# B&R Automation Studio project NAELD004C00R10L518F00 (part 23)

#### Act_Main_Bffr.st
```iecst
(** 2013-05-27 **)
ACTION Act_Main_Bffr:

	CASE usiStep OF
		//Buffer 1
		0:
			eBuffer1Act	:= BufferActCreateDir;

			IF (p_eBuffer1Status = Done) AND (p_eBuffer1Stat = BufferActCreateDir) THEN

				eBuffer1Act	:= BufferActIdle;
				usiStep		:= 1;

			ELSIF p_eBuffer1Status = Error THEN

				eBuffer1Act	:= BufferActIdle;
				usiStep		:= 10;

			END_IF

		1:
			eBuffer1Act	:= BufferActBGStartBffrSetFull;		//BufferActBGStartBffrSetMty

			IF (p_eBuffer1Status = Done) AND (p_eBuffer1Stat = BufferActBGStartBffrSetFull) THEN		//BufferActBGStartBffrSetMty

				eBuffer1Act	:= BufferActIdle;
				usiStep		:= 2;

			ELSIF p_eBuffer1Status = Error THEN

				eBuffer1Act	:= BufferActIdle;
				usiStep		:= 10;

			END_IF

		2:
			IF p_bMagPresent1 = FALSE AND p_bMagPresentSensor1 = TRUE THEN
				usiStep	:= 4;
			ELSE
				usiStep	:= 3;
			END_IF

		3:
			eBuffer1Act	:= BufferActBGStartUpdtSen;

			IF (p_eBuffer1Status = Done) AND (p_eBuffer1Stat = BufferActBGStartUpdtSen) THEN

				eBuffer1Act	:= BufferActIdle;
				usiStep		:= 5;

			ELSIF p_eBuffer1Status = Error THEN

				eBuffer1Act	:= BufferActIdle;
				usiStep		:= 10;

			END_IF

		4:
			eBuffer1Act	:= BufferActBGStartUpdtSen;

			IF (p_eBuffer1Status = Done) AND (p_eBuffer1Stat = BufferActBGStartUpdtSen) THEN

				eBuffer1Act	:= BufferActIdle;
				usiStep		:= 6;

			ELSIF p_eBuffer1Status = Error THEN

				eBuffer1Act	:= BufferActIdle;
				usiStep		:= 10;

			END_IF

		5:
			eBuffer1Act	:= BufferActGetRetainBffr;

			IF (p_eBuffer1Status = Done) AND (p_eBuffer1Stat = BufferActGetRetainBffr) THEN

				eBuffer1Act	:= BufferActIdle;
				usiStep		:= 7;

			ELSIF p_eBuffer1Status = Error THEN

				eBuffer1Act	:= BufferActIdle;
				usiStep		:= 10;

			END_IF

		6:
			eBuffer1Act	:= BufferActSetFull;		//BufferActSetMty

			IF (p_eBuffer1Status = Done) AND (p_eBuffer1Stat = BufferActSetFull) THEN		//BufferActSetMty

				eBuffer1Act	:= BufferActIdle;
				usiStep		:= 7;

			ELSIF p_eBuffer1Status = Error THEN

				eBuffer1Act	:= BufferActIdle;
				usiStep		:= 10;

			END_IF

		7:
			eBuffer1Act	:= BufferActBGStartCoolFan;

			IF (p_eBuffer1Status = Done) AND (p_eBuffer1Stat = BufferActBGStartCoolFan) THEN

				eBuffer1Act		:= BufferActIdle;
				usiStep			:= 10;

			ELSIF p_eBuffer1Status = Error THEN

				eBuffer1Act		:= BufferActIdle;
				usiStep			:= 10;

			END_IF

		//Buffer 2
		10:
			eBuffer2Act	:= BufferActCreateDir;

			IF (p_eBuffer2Status = Done) AND (p_eBuffer2Stat = BufferActCreateDir) THEN

				eBuffer2Act	:= BufferActIdle;
				usiStep		:= 11;

			ELSIF p_eBuffer2Status = Error THEN

				eBuffer2Act	:= BufferActIdle;
				usiStep		:= 20;

			END_IF

		11:
			eBuffer2Act	:= BufferActBGStartBffrSetFull;		//BufferActBGStartBffrSetMty

			IF (p_eBuffer2Status = Done) AND (p_eBuffer2Stat = BufferActBGStartBffrSetFull) THEN		//BufferActBGStartBffrSetMty

				eBuffer2Act	:= BufferActIdle;
				usiStep		:= 12;

			ELSIF p_eBuffer2Status = Error THEN

				eBuffer2Act	:= BufferActIdle;
				usiStep		:= 20;

			END_IF

		12:
			IF p_bMagPresent2 = FALSE AND p_bMagPresentSensor2 = TRUE THEN
				usiStep	:= 14;
			ELSE
				usiStep	:= 13;
			END_IF

		13:
			eBuffer2Act	:= BufferActBGStartUpdtSen;

			IF (p_eBuffer2Status = Done) AND (p_eBuffer2Stat = BufferActBGStartUpdtSen) THEN

				eBuffer2Act	:= BufferActIdle;
				usiStep		:= 15;

			ELSIF p_eBuffer2Status = Error THEN

				eBuffer2Act	:= BufferActIdle;
				usiStep		:= 20;

			END_IF

		14:
			eBuffer2Act	:= BufferActBGStartUpdtSen;

			IF (p_eBuffer2Status = Done) AND (p_eBuffer2Stat = BufferActBGStartUpdtSen) THEN

				eBuffer2Act	:= BufferActIdle;
				usiStep		:= 16;

			ELSIF p_eBuffer2Status = Error THEN

				eBuffer2Act	:= BufferActIdle;
				usiStep		:= 20;

			END_IF

		15:
			eBuffer2Act	:= BufferActGetRetainBffr;

			IF (p_eBuffer2Status = Done) AND (p_eBuffer2Stat = BufferActGetRetainBffr) THEN

				eBuffer2Act	:= BufferActIdle;
				usiStep		:= 17;

			ELSIF p_eBuffer2Status = Error THEN

				eBuffer2Act	:= BufferActIdle;
				usiStep		:= 20;

			END_IF

		16:
			eBuffer2Act	:= BufferActSetFull;		//BufferActSetMty

			IF (p_eBuffer2Status = Done) AND (p_eBuffer2Stat = BufferActSetFull) THEN		//BufferActSetMty

				eBuffer2Act	:= BufferActIdle;
				usiStep		:= 17;

			ELSIF p_eBuffer2Status = Error THEN

				eBuffer2Act	:= BufferActIdle;
				usiStep		:= 20;

			END_IF

		17:
			eBuffer2Act	:= BufferActBGStartCoolFan;

			IF (p_eBuffer2Status = Done) AND (p_eBuffer2Stat = BufferActBGStartCoolFan) THEN

				eBuffer2Act		:= BufferActIdle;
				usiStep			:= 20;

			ELSIF p_eBuffer2Status = Error THEN

				eBuffer2Act		:= BufferActIdle;
				usiStep			:= 20;

			END_IF

		//Buffer 3
		20:
			eBuffer3Act	:= BufferActCreateDir;

			IF (p_eBuffer3Status = Done) AND (p_eBuffer3Stat = BufferActCreateDir) THEN

				eBuffer3Act		:= BufferActIdle;
				usiStep			:= 21;

			ELSIF p_eBuffer3Status = Error THEN

				eBuffer3Act		:= BufferActIdle;
				usiStep			:= 30;

			END_IF

		21:
			eBuffer3Act	:= BufferActBGStartBffrSetFull;		//BufferActBGStartBffrSetMty

			IF (p_eBuffer3Status = Done) AND (p_eBuffer3Stat = BufferActBGStartBffrSetFull) THEN		//BufferActBGStartBffrSetMty

				eBuffer3Act		:= BufferActIdle;
				usiStep			:= 22;

			ELSIF p_eBuffer3Status = Error THEN

				eBuffer3Act		:= BufferActIdle;
				usiStep			:= 30;

			END_IF

		22:
			IF p_bMagPresent3 = FALSE AND p_bMagPresentSensor3 = TRUE THEN
				usiStep	:= 24;
			ELSE
				usiStep	:= 23;
			END_IF

		23:
			eBuffer3Act	:= BufferActBGStartUpdtSen;

			IF (p_eBuffer3Status = Done) AND (p_eBuffer3Stat = BufferActBGStartUpdtSen) THEN

				eBuffer3Act		:= BufferActIdle;
				usiStep			:= 25;

			ELSIF p_eBuffer3Status = Error THEN

				eBuffer3Act		:= BufferActIdle;
				usiStep			:= 30;

			END_IF

		24:
			eBuffer3Act	:= BufferActBGStartUpdtSen;

			IF (p_eBuffer3Status = Done) AND (p_eBuffer3Stat = BufferActBGStartUpdtSen) THEN

				eBuffer3Act		:= BufferActIdle;
				usiStep			:= 26;

			ELSIF p_eBuffer3Status = Error THEN

				eBuffer3Act		:= BufferActIdle;
				usiStep			:= 30;

			END_IF

		25:
			eBuffer3Act	:= BufferActGetRetainBffr;

			IF (p_eBuffer3Status = Done) AND (p_eBuffer3Stat = BufferActGetRetainBffr) THEN

				eBuffer3Act		:= BufferActIdle;
				usiStep			:= 27;

			ELSIF p_eBuffer3Status = Error THEN

				eBuffer3Act		:= BufferActIdle;
				usiStep			:= 30;

			END_IF

		26:
			eBuffer3Act	:= BufferActSetFull;		//BufferActSetMty

			IF (p_eBuffer3Status = Done) AND (p_eBuffer3Stat = BufferActSetFull) THEN		//BufferActSetMty

				eBuffer3Act		:= BufferActIdle;
				usiStep			:= 27;

			ELSIF p_eBuffer3Status = Error THEN

				eBuffer3Act		:= BufferActIdle;
				usiStep			:= 30;

			END_IF

		27:
			eBuffer3Act	:= BufferActBGStartCoolFan;

			IF (p_eBuffer3Status = Done) AND (p_eBuffer3Stat = BufferActBGStartCoolFan) THEN

				eBuffer3Act		:= BufferActIdle;
				usiStep			:= 30;

			ELSIF p_eBuffer3Status = Error THEN

				eBuffer3Act		:= BufferActIdle;
				usiStep			:= 30;

			END_IF

			//Buffer 4
		30:
			eBuffer4Act	:= BufferActCreateDir;

			IF (p_eBuffer4Status = Done) AND (p_eBuffer4Stat = BufferActCreateDir) THEN

				eBuffer4Act		:= BufferActIdle;
				usiStep			:= 31;

			ELSIF p_eBuffer4Status = Error THEN

				eBuffer4Act		:= BufferActIdle;
				usiStep			:= 0;
				eStartupStep1	:= StartupStepAlarm;

			END_IF

		31:
			eBuffer4Act	:= BufferActBGStartBffrSetFull;		//BufferActBGStartBffrSetMty

			IF (p_eBuffer4Status = Done) AND (p_eBuffer4Stat = BufferActBGStartBffrSetFull) THEN		//BufferActBGStartBffrSetMty

				eBuffer4Act		:= BufferActIdle;
				usiStep			:= 32;

			ELSIF p_eBuffer4Status = Error THEN

				eBuffer4Act		:= BufferActIdle;
				usiStep			:= 0;
				eStartupStep1	:= StartupStepAlarm;

			END_IF

		32:
			IF p_bMagPresent4 = FALSE AND p_bMagPresentSensor4 = TRUE THEN
				usiStep	:= 34;
			ELSE
				usiStep	:= 33;
			END_IF

		33:
			eBuffer4Act	:= BufferActBGStartUpdtSen;

			IF (p_eBuffer4Status = Done) AND (p_eBuffer4Stat = BufferActBGStartUpdtSen) THEN

				eBuffer4Act		:= BufferActIdle;
				usiStep			:= 35;

			ELSIF p_eBuffer4Status = Error THEN

				eBuffer4Act		:= BufferActIdle;
				usiStep			:= 0;
				eStartupStep1	:= StartupStepAlarm;

			END_IF

		34:
			eBuffer4Act	:= BufferActBGStartUpdtSen;

			IF (p_eBuffer4Status = Done) AND (p_eBuffer4Stat = BufferActBGStartUpdtSen) THEN

				eBuffer4Act		:= BufferActIdle;
				usiStep			:= 36;

			ELSIF p_eBuffer4Status = Error THEN

				eBuffer4Act		:= BufferActIdle;
				usiStep			:= 0;
				eStartupStep1	:= StartupStepAlarm;

			END_IF

		35:
			eBuffer4Act	:= BufferActGetRetainBffr;

			IF (p_eBuffer4Status = Done) AND (p_eBuffer4Stat = BufferActGetRetainBffr) THEN

				eBuffer4Act		:= BufferActIdle;
				usiStep			:= 37;

			ELSIF p_eBuffer4Status = Error THEN

				eBuffer4Act		:= BufferActIdle;
				usiStep			:= 0;
				eStartupStep1	:= StartupStepAlarm;

			END_IF

		36:
			eBuffer4Act	:= BufferActSetFull;		//BufferActSetMty

			IF (p_eBuffer4Status = Done) AND (p_eBuffer4Stat = BufferActSetFull) THEN		//BufferActSetMty

				eBuffer4Act		:= BufferActIdle;
				usiStep			:= 37;

			ELSIF p_eBuffer4Status = Error THEN

				eBuffer4Act		:= BufferActIdle;
				usiStep			:= 0;
				eStartupStep1	:= StartupStepAlarm;

			END_IF

		37:
			eBuffer4Act	:= BufferActBGStartCoolFan;

			IF (p_eBuffer4Status = Done) AND (p_eBuffer4Stat = BufferActBGStartCoolFan) THEN

				eBuffer4Act		:= BufferActIdle;
				usiStep			:= 0;
				eStartupStep1	:= StartupStepAlarm;

			ELSIF p_eBuffer4Status = Error THEN

				eBuffer4Act		:= BufferActIdle;
				usiStep			:= 0;
				eStartupStep1	:= StartupStepAlarm;

			END_IF
	END_CASE

END_ACTION
```

#### Act_Main_Alarm.st
```iecst
(** 2019-03-28 **)
ACTION Act_Main_Alarm:

	CASE usiStep OF
		0:
			eAlarmAct	:= AlarmActCreateDir;

			IF (p_eAlarmStatus = Done) AND (p_eAlarmStat = AlarmActCreateDir) THEN

				eAlarmAct		:= AlarmActIdle;
				usiStep			:= 1;

			ELSIF p_eAlarmStatus = Error THEN

				eAlarmAct		:= AlarmActIdle;
				usiStep			:= 0;
		//		eStartupStep1	:= StartupStepHermes;
				eStartupStep1	:= StartupStepSerial;
			END_IF

		1:
			eAlarmAct	:= AlarmActDeleteOldLog;

			IF (p_eAlarmStatus = Done) AND (p_eAlarmStat = AlarmActDeleteOldLog) THEN

				eAlarmAct		:= AlarmActIdle;
				usiStep			:= 2;

			ELSIF p_eAlarmStatus = Error THEN

				eAlarmAct		:= AlarmActIdle;
				usiStep			:= 0;
		//		eStartupStep1	:= StartupStepHermes;
				eStartupStep1	:= StartupStepSerial;
			END_IF

		2:
			eAlarmAct	:= AlarmActReadHistory;

			IF (p_eAlarmStatus = Done) AND (p_eAlarmStat = AlarmActReadHistory) THEN

				eAlarmAct		:= AlarmActIdle;
				usiStep			:= 3;

			ELSIF p_eAlarmStatus = Error THEN

				eAlarmAct		:= AlarmActIdle;
				usiStep			:= 0;
		//		eStartupStep1	:= StartupStepHermes;
				eStartupStep1	:= StartupStepSerial;
			END_IF

		3:
			eAlarmAct	:= AlarmActBGStartLog;

			IF (p_eAlarmStatus = Done) AND (p_eAlarmStat = AlarmActBGStartLog) THEN

				eAlarmAct		:= AlarmActIdle;
				usiStep			:= 0;
		//		eStartupStep1	:= StartupStepHermes;
				eStartupStep1	:= StartupStepSerial;
			ELSIF p_eAlarmStatus = Error THEN

				eAlarmAct		:= AlarmActIdle;
				usiStep			:= 0;
		//		eStartupStep1	:= StartupStepHermes;
				eStartupStep1	:= StartupStepSerial;
			END_IF

	END_CASE

END_ACTION
```

#### Act_Main_Serial.st
```iecst
(** 2019-03-28 **)
ACTION Act_Main_Serial:

	CASE usiStep OF
		0:
			eFrmAct	:= FrmActCreateDir;

			IF (p_eFrmStatus = Done) AND (p_eFrmStat = FrmActCreateDir)THEN

				eFrmAct		:= FrmActIdle;
				usiStep			:= 1;

			ELSIF p_eFrmStatus = Error THEN

				eFrmAct			:= FrmActIdle;
				usiStep			:= 1;
				eStartupStep1	:= StartupStepHermes;

			END_IF

		1:
			eFrmAct	:= FrmActDeleteOldLog;

			IF (p_eFrmStatus = Done) AND (p_eFrmStat = FrmActDeleteOldLog) THEN

				eFrmAct			:= FrmActIdle;
				usiStep			:= 2;

			ELSIF p_eFrmStatus = Error THEN

				eFrmAct			:= FrmActIdle;
				usiStep			:= 2;
				eStartupStep1	:= StartupStepHermes;

			END_IF

		2:
			eUSBAct	:= USBRdrActCreateDir;
			IF (p_eUSBStatus = Done) AND (p_eUSBStat = USBRdrActCreateDir) THEN
				eUSBAct		:= USBRdrActIdle;
				usiStep			:= 3;

			ELSIF  p_eUSBStatus = Error THEN
				eUSBAct			:= USBRdrActIdle;
				usiStep			:= 3;
			END_IF

		3:
			eUSBAct	:= USBRdrActDeleteOldLog;
			IF (p_eUSBStatus = Done) AND (p_eUSBStat = USBRdrActDeleteOldLog)THEN
				eUSBAct			:= USBRdrActIdle;
				usiStep			:= 0;
				eStartupStep1	:= StartupStepHermes;

			ELSIF p_eUSBStatus = Error THEN

				eUSBAct			:= USBRdrActIdle;
				usiStep			:= 0;
				eStartupStep1	:= StartupStepHermes;

			END_IF
	END_CASE

END_ACTION
```

#### Act_Main_Hermes.st
```iecst
(** 2019-05-04 **)
ACTION Act_Main_Hermes:

	CASE usiStep OF
		0:
			eHermesAct	:= HermesActCreateDir;

			IF (p_eHermesStatus = Done) AND (p_eHermesStat = HermesActCreateDir) THEN

				eHermesAct		:= HermesActIdle;
				usiStep			:= 1;

			ELSIF p_eHermesStatus = Error THEN

				eHermesAct		:= HermesActIdle;
				usiStep			:= 10;

			END_IF

		1:
			eHermesAct	:= HermesActReadRetain;

			IF (p_eHermesStatus = Done) AND (p_eHermesStat = HermesActReadRetain) THEN

				eHermesAct		:= HermesActIdle;
				usiStep			:= 2;

			ELSIF p_eHermesStatus = Error THEN

				eHermesAct		:= HermesActIdle;
				usiStep			:= 10;

			END_IF

		2:
			eHermesAct	:= HermesActReadConfig;

			IF (p_eHermesStatus = Done) AND (p_eHermesStat = HermesActReadConfig) THEN

				eHermesAct		:= HermesActIdle;
				usiStep			:= 10;

			ELSIF p_eHermesStatus = Error THEN

				eHermesAct		:= HermesActIdle;
				usiStep			:= 10;

			END_IF

		10:
			eRmtHermesAct	:= HermesActDeleteOldLog;

			IF (p_eRmtHermesStatus = Done) AND (p_eRmtHermesStat = HermesActDeleteOldLog) THEN

				eRmtHermesAct	:= HermesActIdle;
				usiStep			:= 11;

			ELSIF p_eRmtHermesStatus = Error THEN

				eRmtHermesAct	:= HermesActIdle;
				usiStep			:= 20;

			END_IF

		11:
			eRmtHermesAct	:= HermesActReadConfig;

			IF (p_eRmtHermesStatus = Done) AND (p_eRmtHermesStat = HermesActReadConfig) THEN

				eRmtHermesAct	:= HermesActIdle;
				usiStep			:= 20;

			ELSIF p_eRmtHermesStatus = Error THEN

				eRmtHermesAct	:= HermesActIdle;
				usiStep			:= 20;

			END_IF

		20:
			eDSHermesAAct	:= HermesActDeleteOldLog;

			IF (p_eDSHermesAStatus = Done) AND (p_eDSHermesAStat = HermesActDeleteOldLog) THEN

				eDSHermesAAct	:= HermesActIdle;
				usiStep			:= 30;

			ELSIF p_eDSHermesAStatus = Error THEN

				eDSHermesAAct	:= HermesActIdle;
				usiStep			:= 30;

			END_IF

		30:
			eDSHermesBAct	:= HermesActDeleteOldLog;

			IF (p_eDSHermesBStatus = Done) AND (p_eDSHermesBStat = HermesActDeleteOldLog) THEN

				eDSHermesBAct	:= HermesActIdle;
				usiStep			:= 0;
			//	eStartupStep1	:= StartupStepSDOWrite;
				eStartupStep1	:= StartupStepSetupUI;

			ELSIF p_eDSHermesBStatus = Error THEN

				eDSHermesBAct	:= HermesActIdle;
				usiStep			:= 0;
			//	eStartupStep1	:= StartupStepSDOWrite;
				eStartupStep1	:= StartupStepSetupUI;

			END_IF

	END_CASE

END_ACTION
```

#### Act_Main_SDOWrite.st
```iecst
(** 2019-10-21 **)
ACTION Act_Main_SDOWrite:

	CASE usiStep OF

		0:
			eAWPushPulAct	:= AWActBGStartModOKChk;

			IF (p_eAWPushOrPullerStatus = Done) AND (p_eAWPushOrPullerStat = AWActBGStartModOKChk) THEN

				eAWPushPulAct	:= AWActIdle;
				usiStep		:= 5;

			ELSIF p_eAWPushOrPullerStatus = Error THEN

				eAWPushPulAct		:= AWActIdle;
				usiStep		:= 5;

			END_IF

		5:
			eAWAct	:= AWActBGStartModOKChk;

			IF (p_eAWStatus = Done) AND (p_eAWStat = AWActBGStartModOKChk) THEN

				eAWAct		:= AWActIdle;
				usiStep		:= 10;

			ELSIF p_eAWStatus = Error THEN

				eAWAct		:= AWActIdle;
				usiStep		:= 10;

			END_IF

		10:
			eServoPPAct	:= PPActBGStartModOKChk;

			IF (p_eServoPPStatus = Done) AND (p_eServoPPStat = PPActBGStartModOKChk) THEN

				eServoPPAct	:= PPActIdle;
				usiStep		:= 15;

			ELSIF p_eServoPPStatus = Error THEN

				eServoPPAct	:= PPActIdle;
				usiStep		:= 15;

			END_IF

		15:
			eTravAct	:= TravActBGStartModOKChk;

			IF (p_eTravStatus = Done) AND (p_eTravStat = TravActBGStartModOKChk) THEN

				eTravAct	:= TravActIdle;
				usiStep		:= 20;

			ELSIF p_eTravStatus = Error THEN

				eTravAct	:= TravActIdle;
				usiStep		:= 20;

			END_IF

		20:
			eLifterAct	:= LifterActBGStartModOKChk;

			IF (p_eLifterStatus = Done) AND (p_eLifterStat = LifterActBGStartModOKChk) THEN

				eLifterAct		:= LifterActIdle;
				usiStep			:= 0;
				eStartupStep1	:= StartupStepSetupUI;

			ELSIF p_eLifterStatus = Error THEN

				eLifterAct		:= LifterActIdle;
				usiStep			:= 0;
				eStartupStep1	:= StartupStepSetupUI;

			END_IF

	END_CASE

END_ACTION
```

### Program Logical/UsrFolder/UsrFolder

#### Local.var
```iecst
(*2019-05-09*)
(**)
(*Local Action, State & Status*)
VAR
	eAct : eUsrFolderAction := UsrFolderActIdle;
	eStat : eUsrFolderAction := UsrFolderActIdle;
	eStatus : eFBStatus := Idle;
	udiStatus : UDINT := 0;
	sStatTxt : STRING[200] := '';
	a_sStatText : ARRAY[0..50] OF STRING[200] := ['Idling','Creating User Directory','Creating Private Directory','Creating Log Directory','Creating LCS Directory',46('')];
END_VAR
(**)
(*Local Alarm*)
VAR
	tyAlmData : tyAlmDat;
	a_tyAlmText : ARRAY[10000..10099] OF tyAlmTxt := [(sAlmText:='Creating User Directory Error',sRcyText:='An Error Occured While Attempting To Create User Directory. Please Contact Nutek For A Possible Solution'),(sAlmText:='Creating Private Directory Error',sRcyText:='An Error Occured While Attempting To Create Private Directory. Please Contact Nutek For A Possible Solution'),(sAlmText:='Creating Log Directory Error',sRcyText:='An Error Occured While Attempting To Create Log Directory. Please Contact Nutek For A Possible Solution'),(sAlmText:='Creating LCS Directory Error',sRcyText:='An Error Occured While Attempting To Create LCS Directory. Please Contact Nutek For A Possible Solution'),96(0)];
END_VAR
(**)
(*Local Output*)
(**)
(*Local Input*)
VAR
	udiRstErr : UDINT := 0;
	sProgNm : STRING[15] := 'UsrFolder';
END_VAR
(**)
(*Local*)
VAR
	bRstErr : BOOL;
	udiRstErrOld : UDINT;
	bInitDone : BOOL;
	bInitialDone : BOOL;
	fbDirCreate1 : fbDirCreate;
	fbDirCreate2 : fbDirCreate;
	fbDirCreate3 : fbDirCreate;
	fbDirCreate4 : fbDirCreate;
	udiModuleNum : UDINT := 5551;
END_VAR
```

#### Act_Alarm.st
```iecst
(** 2019-03-25 **)
ACTION Act_Alarm:

	//Error
	IF EDGEPOS(eStatus = Error) THEN

		tyAlmData.sProgNm		:= p_sProgNm;
		tyAlmData.udiCode		:= udiStatus;
		tyAlmData.eSeverity		:= AlmSeverityError;
		tyAlmData.udiRunTime	:= tyAlmData.udiRunTime + 1;
		tyAlmData.bAlm			:= TRUE;
		tyAlmData.udiModuleNum  := udiModuleNum;
		g_sUsrFolderProgNm		:= p_sProgNm;
		//Get Error Message
		IF tyAlmData.udiCode < 10000 OR tyAlmData.udiCode > 10099 THEN
			tyAlmData.sAlmMsg	:= 'Unknown';
			tyAlmData.sRcyMsg	:= 'Unknown';
		ELSE
			tyAlmData.sAlmMsg	:= a_tyAlmText[tyAlmData.udiCode].sAlmText;
			tyAlmData.sRcyMsg	:= a_tyAlmText[tyAlmData.udiCode].sRcyText;
		END_IF

		sStatTxt	:= tyAlmData.sAlmMsg;

	ELSIF bRstErr AND (tyAlmData.udiCode <> 0) THEN

		tyAlmData.udiCode	:= 0;
		tyAlmData.eSeverity	:= AlmSeverityNA;
		tyAlmData.sAlmMsg	:= '';
		tyAlmData.sRcyMsg	:= '';
		tyAlmData.bAlm			:= FALSE;
		sStatTxt	:= a_sStatText[eStat];

	END_IF

END_ACTION
```

### Program Logical/LibVer/LibVer

#### Act_Alarm.st
```iecst
(** 2019-03-25 **)
ACTION Act_Alarm:

	//Error
	IF EDGEPOS(eStatus = Error) THEN

		tyAlmData.sProgNm		:= p_sProgNm;
		tyAlmData.udiCode		:= udiStatus;
		tyAlmData.udiRunTime	:= tyAlmData.udiRunTime + 1;

		tyAlmData.udiModuleNum  := udiModuleNum;
		g_sLibVerProgNm			:= p_sProgNm;

		IF tyAlmData.udiCode = 10012 THEN
			tyAlmData.eSeverity	:= AlmSeverityWarning;
			tyAlmData.bWarning		:= TRUE;
			//Get Error Message
			tyAlmData.sAlmMsg	:= a_tyAlmText[tyAlmData.udiCode].sAlmText;

			FOR di := 0 TO c_diLibNum DO
				IF a_bVerMismatch[di] = TRUE THEN
					tyAlmData.sAlmMsg	:= CONCAT(tyAlmData.sAlmMsg , ' (');
					tyAlmData.sAlmMsg	:= CONCAT(tyAlmData.sAlmMsg , a_tyInfoOut[di].sName);
					tyAlmData.sAlmMsg	:= CONCAT(tyAlmData.sAlmMsg , ')');
					g_sLiberWarnName    := a_tyInfoOut[di].sName;
					EXIT;
				END_IF
			END_FOR

			tyAlmData.sRcyMsg	:= a_tyAlmText[tyAlmData.udiCode].sRcyText;

		ELSE
			tyAlmData.eSeverity	:= AlmSeverityError;
			tyAlmData.bAlm		:= TRUE;
			//Get Error Message
			IF tyAlmData.udiCode < 10000 OR tyAlmData.udiCode > 10099 THEN
				tyAlmData.sAlmMsg	:= 'Unknown';
				tyAlmData.sRcyMsg	:= 'Unknown';
			ELSE
				tyAlmData.sAlmMsg	:= a_tyAlmText[tyAlmData.udiCode].sAlmText;
				tyAlmData.sRcyMsg	:= a_tyAlmText[tyAlmData.udiCode].sRcyText;
			END_IF

			sStatTxt	:= tyAlmData.sAlmMsg;

		END_IF

	ELSIF bRstErr AND (tyAlmData.udiCode <> 0) THEN

		tyAlmData.udiCode	:= 0;
		tyAlmData.eSeverity	:= AlmSeverityNA;
		tyAlmData.sAlmMsg	:= '';
		tyAlmData.sRcyMsg	:= '';
		tyAlmData.bAlm			:= FALSE;
		tyAlmData.bWarning		:= FALSE;
		sStatTxt	:= a_sStatText[eStat];

	END_IF

END_ACTION
```

### Program Logical/Time/Time

#### Act_Alarm.st
```iecst
(** 2019-03-25 **)
ACTION Act_Alarm:

	//Error
	IF EDGEPOS(eStatus = Error) THEN

		tyAlmData.sProgNm		:= p_sProgNm;
		tyAlmData.udiCode		:= udiStatus;
		tyAlmData.eSeverity		:= AlmSeverityError;
		tyAlmData.udiRunTime	:= tyAlmData.udiRunTime + 1;
		tyAlmData.bAlm			:= TRUE;
		tyAlmData.udiModuleNum  := udiModuleNum;
		g_sTimeProgNm			:= p_sProgNm;
		//Get Error Message
		IF tyAlmData.udiCode < 10000 OR tyAlmData.udiCode > 10099 THEN
			tyAlmData.sAlmMsg	:= 'Unknown';
			tyAlmData.sRcyMsg	:= 'Unknown';
		ELSE
			tyAlmData.sAlmMsg	:= a_tyAlmText[tyAlmData.udiCode].sAlmText;
			tyAlmData.sRcyMsg	:= a_tyAlmText[tyAlmData.udiCode].sRcyText;
		END_IF

		sStatTxt	:= tyAlmData.sAlmMsg;

	ELSIF bRstErr AND (tyAlmData.udiCode <> 0) THEN

		tyAlmData.udiCode	:= 0;
		tyAlmData.eSeverity	:= AlmSeverityNA;
		tyAlmData.sAlmMsg	:= '';
		tyAlmData.sRcyMsg	:= '';
		tyAlmData.bAlm			:= FALSE;
		sStatTxt	:= a_sStatText[eStat];

	END_IF

END_ACTION
```

#### Act_Alarm1.st
```iecst
(** 2019-03-25 **)
ACTION Act_Alarm1:

	//Error
	IF EDGEPOS(eStatus1 = Error) THEN

		tyAlmData1.sProgNm		:= p_sProgNm;
		tyAlmData1.udiCode		:= udiStatus1;
		tyAlmData1.eSeverity	:= AlmSeverityError;
		tyAlmData1.udiRunTime	:= tyAlmData1.udiRunTime + 1;
		tyAlmData1.bAlm			:= TRUE;
		tyAlmData1.udiModuleNum  := udiModuleNum;
		g_sTimeProgNm			:= p_sProgNm;
		//Get Error Message
		IF tyAlmData1.udiCode < 10000 OR tyAlmData1.udiCode > 10099 THEN
			tyAlmData1.sAlmMsg	:= 'Unknown';
			tyAlmData1.sRcyMsg	:= 'Unknown';
		ELSE
			tyAlmData1.sAlmMsg	:= a_tyAlmText[tyAlmData1.udiCode].sAlmText;
			tyAlmData1.sRcyMsg	:= a_tyAlmText[tyAlmData1.udiCode].sRcyText;
		END_IF

		sStatTxt	:= tyAlmData1.sAlmMsg;

	ELSIF bRstErr AND (tyAlmData1.udiCode <> 0) THEN

		tyAlmData1.udiCode		:= 0;
		tyAlmData1.eSeverity	:= AlmSeverityNA;
		tyAlmData1.sAlmMsg		:= '';
		tyAlmData1.sRcyMsg		:= '';
		tyAlmData1.bAlm			:= FALSE;
		sStatTxt	:= a_sStatText[eStat];

	END_IF

END_ACTION
```

### HWInfo.typ
```iecst
(*2020-09-22*)
(**)
(*Action*)

TYPE
	eHWInfoAction :
		(
		HWInfoActIdle,
		HWInfoActGetIPAddr,
		HWInfoActGetSubnetMask,
		HWInfoActGetMacAddr,
		HWInfoActSetIPAddr,
		HWInfoActSetSubnetMask,
		HWInfoActGetEthConfigMode,
		HWInfoActSetEthConfigMode
		);
	eNetworkConfigMod :
		(
		SetIPManually := 0,
		IPFromDHCPServer := 1
		);
END_TYPE
```

### Program Logical/HWInfo/HWInfo

#### Local.var
```iecst
(*2020-10-05*)
(**)
(*Local Action, State & Status*)
VAR
	eAct : eHWInfoAction := HWInfoActIdle;
	eStat : eHWInfoAction := HWInfoActIdle;
	eStatus : eFBStatus := Idle;
	udiStatus : UDINT := 0;
	sStatTxt : STRING[200] := '';
	a_sStatText : ARRAY[0..50] OF STRING[200] := ['Idling','Get IP Address','Get IP Subnet Mask','Get Mac Address','Setting IP Address','Setting IP Subnet Mask',45('')];
END_VAR
(**)
(*Local Alarm*)
VAR
	tyAlmData : tyAlmDat;
	a_tyAlmText : ARRAY[10000..10099] OF tyAlmTxt := [(sAlmText:='Get IP Address Error',sRcyText:='Failed To Obtain The IP Address. Please Contact Nutek For A Possible Solution.'),(sAlmText:='Get Subnet Mask Error',sRcyText:='Failed To Obtain The Subnet Mask. Please Contact Nutek For A Possible Solution.'),(sAlmText:='Get Mac Address Error',sRcyText:='Failed To Obtain The Mac Address. Please Contact Nutek For A Possible Solution.'),(sAlmText:='Set IP Address Error',sRcyText:='Invalid IP Address Configuration. Please Contact Nutek For A Possible Solution.'),(sAlmText:='Set Subnet Mask Error',sRcyText:='Invalid Subnet Mask Configuration. Please Contact Nutek For A Possible Solution.'),(sAlmText:='Get Network Configuration Mode Error',sRcyText:='Failed To Obtain The Network Configuration. Please Contact Nutek For A Possible Solution.'),(sAlmText:='Set Network Configuration Mode Error',sRcyText:='Invalid Network Configuration . Please Contact Nutek For A Possible Solution.'),93(0)];
END_VAR
(**)
(*Local Output*)
VAR
	sIPAddr : STRING[15];
	sSubnetMask : STRING[15];
	a_usiMacAddr : ARRAY[0..5] OF USINT;
	udiConfigMode : UDINT;
END_VAR
(**)
(*Local Input*)
VAR
	udiRstErr : UDINT := 0;
	sSetIPAddr : STRING[15];
	sSetSubnetMask : STRING[15];
	sDevice : STRING[3] := 'IF2';
	sProgNm : STRING[15] := 'HWInfo';
	bNtSettingsLoadDone : BOOL := TRUE;
	usiNetworkMode : USINT;
END_VAR
(**)
(*Local*)
VAR
	bRstErr : BOOL;
	udiRstErrOld : UDINT;
	bInitDone : BOOL;
	bInitialDone : BOOL;
	fbGetIPAddr : CfgGetIPAddr;
	fbGetSubnetMask : CfgGetSubnetMask;
	fbGetMacAddr : CfgGetMacAddr;
	fbSetIPAddr : CfgSetIPAddr;
	fbSetSubnetMask : CfgSetSubnetMask;
	fbSetETHConfigMode : CfgSetEthConfigMode;
	fbGetETHConfigMode : CfgGetEthConfigMode;
	usiInitialFile : USINT;
	a_sMacAddr : ARRAY[0..5] OF STRING[3];
	sMacAddr : STRING[25];
	usi : USINT;
	fbFileFullWrite_0 : fbFileFullWrite;
	udiModuleNum : UDINT := 5651;
END_VAR
```

#### Act_InitGlobal.st
```iecst
(** 2020-09-22 **)
ACTION Act_InitGlobal:

	(* Always Change If Project Change *)

	//Pass Data To Link
	p_bLinkStartupRun ACCESS p_StartupRun;

	//Pass Data To Internal Use
	p_udiRstErr ACCESS p_RstErrReset;
	p_sSetIPAddr ACCESS p_UISetIPAddr;
	p_sSetSubnetMask ACCESS p_UISetSubnetMask;
	p_sDevice ACCESS p_NtParamHWInfoDevice;
	p_sProgNm ACCESS p_NtParamHWInfoProgNm;
	p_bNtSettingsLoadDone ACCESS p_StartupNtSettingsLoadDone;
	p_usiNetworkMod ACCESS p_UINetworkMode;

	(* Always Change If Project Change *)

END_ACTION
```

#### Act_Main.st
```iecst
(** 2020-10-05 **)
ACTION Act_Main:

	//Main
	CASE eStat OF

		HWInfoActIdle:
			IF eStatus <> Idle THEN	//Reset Data
				//Private
				fbGetIPAddr(enable := FALSE);
				fbGetMacAddr(enable := FALSE);
				fbSetIPAddr(enable := FALSE);
				fbSetSubnetMask(enable := FALSE);
				fbGetETHConfigMode(enable := FALSE);
				fbSetETHConfigMode(enable := FALSE);

				sStatTxt	:= a_sStatText[eStat];

			END_IF

			eStatus	:= Idle;

		HWInfoActGetIPAddr:
			IF eStatus = Idle OR eStatus = Busy THEN

				eStatus	:= Busy;

				sStatTxt	:= a_sStatText[eStat];

				IF DiagCpuIsSimulated() = FALSE THEN
					fbGetIPAddr(enable := TRUE);
					IF fbGetIPAddr.status = 0 THEN
						eStatus	:= Done;
					ELSIF fbGetIPAddr.status < 65534 THEN
						udiStatus	:= 10000;	//Get IP Address Error
						eStatus		:= Error;
					END_IF

				ELSE
					eStatus	:= Done;
					sIPAddr	:= '127.0.0.1';

				END_IF

			END_IF

		HWInfoActGetSubnetMask:
			IF eStatus = Idle OR eStatus = Busy THEN

				eStatus	:= Busy;

				sStatTxt	:= a_sStatText[eStat];

				IF DiagCpuIsSimulated() = FALSE THEN
					fbGetSubnetMask(enable := TRUE);
					IF fbGetSubnetMask.status = 0 THEN
						eStatus	:= Done;
					ELSIF fbGetSubnetMask.status < 65534 THEN
						udiStatus	:= 10001;	//Get Subnet Mask Error
						eStatus		:= Error;
					END_IF

				ELSE
					eStatus		:= Done;
					sSubnetMask	:= '255.255.0.0';

				END_IF

			END_IF

		HWInfoActGetMacAddr:
			IF eStatus = Idle OR eStatus = Busy THEN

				eStatus	:= Busy;

				sStatTxt	:= a_sStatText[eStat];

				IF DiagCpuIsSimulated() = FALSE THEN
					fbGetMacAddr(enable := TRUE);
					IF fbGetMacAddr.status = 0 THEN
						eStatus	:= Done;
					ELSIF fbGetMacAddr.status < 65534 THEN
						udiStatus	:= 10002;	//Get Mac Address Error
						eStatus		:= Error;
					END_IF

				ELSE
					eStatus	:= Done;

				END_IF

			END_IF

		HWInfoActSetIPAddr:
			IF eStatus = Idle OR eStatus = Busy THEN

				eStatus	:= Busy;

				sStatTxt	:= a_sStatText[eStat];

				IF DiagCpuIsSimulated() = FALSE THEN
					fbSetIPAddr(enable := TRUE);
					IF fbSetIPAddr.status = 0 THEN
						sIPAddr	:= p_sSetIPAddr;
						eStatus	:= Done;
					ELSIF fbSetIPAddr.status < 65534 THEN
						udiStatus	:= 10003;	//Set IP Address Error
						eStatus		:= Error;
					END_IF

				ELSE
					eStatus	:= Done;

				END_IF

			END_IF

		HWInfoActSetSubnetMask:
			IF eStatus = Idle OR eStatus = Busy THEN

				eStatus	:= Busy;

				sStatTxt	:= a_sStatText[eStat];

				IF DiagCpuIsSimulated() = FALSE THEN
					fbSetSubnetMask(enable := TRUE);
					IF fbSetSubnetMask.status = 0 THEN
						sSubnetMask	:= p_sSetSubnetMask;
						eStatus		:= Done;
					ELSIF fbSetSubnetMask.status < 65534 THEN
						udiStatus	:= 10004;	//Set Subnet Mask Error
						eStatus		:= Error;
					END_IF

				ELSE
					eStatus	:= Done;

				END_IF

			END_IF

		HWInfoActGetEthConfigMode:
			IF eStatus = Idle OR eStatus = Busy THEN

				eStatus	:= Busy;

				sStatTxt	:= a_sStatText[eStat];
				IF DiagCpuIsSimulated() = FALSE THEN
					fbGetETHConfigMode(enable := TRUE);
					IF fbGetETHConfigMode.status = 0 THEN
						udiConfigMode := fbGetETHConfigMode.ConfigMode;
						eStatus	:= Done;
					ELSIF fbGetETHConfigMode.status < 65534 THEN
						udiStatus	:= 10005;	//Get Network Configuration  Error
						eStatus		:= Error;
					END_IF

				ELSE
					eStatus	:= Done;

				END_IF

			END_IF

		HWInfoActSetEthConfigMode:
			IF eStatus = Idle OR eStatus = Busy THEN

				eStatus	:= Busy;

				sStatTxt	:= a_sStatText[eStat];

				IF DiagCpuIsSimulated() = FALSE THEN
					fbSetETHConfigMode.ConfigMode := USINT_TO_UDINT(p_usiNetworkMod);
					fbSetETHConfigMode(enable := TRUE);

					IF fbSetETHConfigMode.status = 0 THEN
						eStatus	:= Done;
					ELSIF fbSetETHConfigMode.status < 65534 THEN
						udiStatus	:= 10006;	//Set Network Configuration  Error
						eStatus		:= Error;
					END_IF

				ELSE
					eStatus	:= Done;

				END_IF

			END_IF

	END_CASE

	//Generate file
	IF a_usiMacAddr[3] <> 0 AND usiInitialFile <2 THEN
		CASE usi OF
			0:
				FOR usi:= 0 TO 5 DO
					//a_sMacAddr[usi] := USINT_TO_STRING(a_usiMacAddr[usi]);
					sprintf1(ADR(a_sMacAddr[usi]), ADR('%+02x'), a_usiMacAddr[usi]);
				END_FOR
				sMacAddr := CONCAT('PLC= ',CONCAT(a_sMacAddr[0],'-'));
				FOR usi := 1 TO 5 DO
					sMacAddr := CONCAT(CONCAT(sMacAddr,a_sMacAddr[usi]),'-');
				END_FOR
				sMacAddr := DELETE(sMacAddr,1,LEN(sMacAddr));
				usi := 1;
			1:
				fbFileFullWrite_0(bEn := TRUE, sDevice := 'Log', sFile := 'PLC_MacAddress.txt', udiOffset := 0, p_Src := ADR(sMacAddr), udiLen := SIZEOF(sMacAddr), udiOption := 0);
				IF fbFileFullWrite_0.udiStatus = 0 THEN
					fbFileFullWrite_0(bEn := FALSE);
					IF usiInitialFile = 1 THEN
						usi := 0;
					END_IF
					usiInitialFile := usiInitialFile +1;
				END_IF

		END_CASE
	END_IF

END_ACTION
```

### Program Logical/TLBuz/TLBuz

#### InputRef.var
```iecst
(*2020-03-16*)
(**)
(*General*)
VAR
	p_eAct : REFERENCE TO eTLBuzAction;
END_VAR
(**)
(*Configuration*)
VAR
	p_bManual : REFERENCE TO BOOL;
	p_bStartup : REFERENCE TO BOOL;
	p_bErr : REFERENCE TO BOOL;
	p_bErrNoBuz : REFERENCE TO BOOL;
	p_bWarning : REFERENCE TO BOOL;
	p_bWarningNoBuz : REFERENCE TO BOOL;
	p_bWarning1 : REFERENCE TO BOOL;
	p_bWarning1NoBuz : REFERENCE TO BOOL;
	p_bWarning2 : REFERENCE TO BOOL;
	p_bWarning2NoBuz : REFERENCE TO BOOL;
	p_bWarning3 : REFERENCE TO BOOL;
	p_bWarning3NoBuz : REFERENCE TO BOOL;
	p_bWarning4 : REFERENCE TO BOOL;
	p_bWarning4NoBuz : REFERENCE TO BOOL;
	p_bWarning5 : REFERENCE TO BOOL;
	p_bWarning5NoBuz : REFERENCE TO BOOL;
	p_bChgRcp : REFERENCE TO BOOL;
	p_bSeqStop : REFERENCE TO BOOL;
	p_bStep : REFERENCE TO BOOL;
	p_bOps : REFERENCE TO BOOL;
	p_bStandby : REFERENCE TO BOOL;
	p_bSimulation : REFERENCE TO BOOL;
	p_bMuteBuz : REFERENCE TO BOOL;
END_VAR
(*TLBuz ChangeRcp Behaviour*)
VAR
	p_tTLChgRcpBlinkTm : REFERENCE TO TIME;
END_VAR
(*TLBuz Error Behaviour*)
VAR
	p_tTLErrBlinkTm : REFERENCE TO TIME;
	p_tBuzErrOnTm : REFERENCE TO TIME;
	p_tBuzErrRestTm : REFERENCE TO TIME;
	p_usiBuzErrOnCntr : REFERENCE TO USINT;
	p_bBuzErrStopSeqEn : REFERENCE TO BOOL;
	p_usiBuzErrStopSeqCntr : REFERENCE TO USINT;
END_VAR
(*TLBuz Default Warning Behaviour*)
VAR
	p_tTLWarnBlinkTm : REFERENCE TO TIME;
	p_tBuzWarnOnTm : REFERENCE TO TIME;
	p_tBuzWarnRestTm : REFERENCE TO TIME;
	p_usiBuzWarnOnCntr : REFERENCE TO USINT;
	p_bBuzWarnStopSeqEn : REFERENCE TO BOOL;
	p_usiBuzWarnStopSeqCntr : REFERENCE TO USINT;
END_VAR
(*TLBuz Special Warning 1 Behaviour*)
VAR
	p_tTLWarn1BlinkTm : REFERENCE TO TIME;
	p_tBuzWarn1OnTm : REFERENCE TO TIME;
	p_tBuzWarn1RestTm : REFERENCE TO TIME;
	p_usiBuzWarn1OnCntr : REFERENCE TO USINT;
	p_bBuzWarn1StopSeqEn : REFERENCE TO BOOL;
	p_usiBuzWarn1StopSeqCntr : REFERENCE TO USINT;
END_VAR
(*TLBuz Special Warning 2 Behaviour*)
VAR
	p_tTLWarn2BlinkTm : REFERENCE TO TIME;
	p_tBuzWarn2OnTm : REFERENCE TO TIME;
	p_tBuzWarn2RestTm : REFERENCE TO TIME;
	p_usiBuzWarn2OnCntr : REFERENCE TO USINT;
	p_bBuzWarn2StopSeqEn : REFERENCE TO BOOL;
	p_usiBuzWarn2StopSeqCntr : REFERENCE TO USINT;
END_VAR
(*TLBuz Special Warning 3 Behaviour*)
VAR
	p_tTLWarn3BlinkTm : REFERENCE TO TIME;
	p_tBuzWarn3OnTm : REFERENCE TO TIME;
	p_tBuzWarn3RestTm : REFERENCE TO TIME;
	p_usiBuzWarn3OnCntr : REFERENCE TO USINT;
	p_bBuzWarn3StopSeqEn : REFERENCE TO BOOL;
	p_usiBuzWarn3StopSeqCntr : REFERENCE TO USINT;
END_VAR
(*TLBuz Special Warning 4 Behaviour*)
VAR
	p_tTLWarn4BlinkTm : REFERENCE TO TIME;
	p_tBuzWarn4OnTm : REFERENCE TO TIME;
	p_tBuzWarn4RestTm : REFERENCE TO TIME;
	p_usiBuzWarn4OnCntr : REFERENCE TO USINT;
	p_bBuzWarn4StopSeqEn : REFERENCE TO BOOL;
	p_usiBuzWarn4StopSeqCntr : REFERENCE TO USINT;
END_VAR
(*TLBuz Special Warning 5 Behaviour*)
VAR
	p_tTLWarn5BlinkTm : REFERENCE TO TIME;
	p_tBuzWarn5OnTm : REFERENCE TO TIME;
	p_tBuzWarn5RestTm : REFERENCE TO TIME;
	p_usiBuzWarn5OnCntr : REFERENCE TO USINT;
	p_bBuzWarn5StopSeqEn : REFERENCE TO BOOL;
	p_usiBuzWarn5StopSeqCntr : REFERENCE TO USINT;
END_VAR
(*TLBuz Special Buz Behaviour*)
VAR
	p_tBuzAlertOnTm : REFERENCE TO TIME;
	p_tBuzAlertRestTm : REFERENCE TO TIME;
	p_usiBuzAlertOnCntr : REFERENCE TO USINT;
	p_bBuzAlertStopSeqEn : REFERENCE TO BOOL;
	p_usiBuzAlertStopSeqCntr : REFERENCE TO USINT;
END_VAR
(*TLBuz Special Ops TL Behaviour*)
VAR
	p_tTLBlueBlinkTm : REFERENCE TO TIME;
	p_tTLAmberBlinkTm : REFERENCE TO TIME;
	p_tTLWhiteBlinkTm : REFERENCE TO TIME;
	p_tTLRedBlinkTm : REFERENCE TO TIME;
	p_tTLGreenBlinkTm : REFERENCE TO TIME;
END_VAR
(**)
VAR
	p_bCoverSwitchSig : REFERENCE TO BOOL;
	p_eTLBuzMode : REFERENCE TO eTLBuzMod;
	p_bAOIErrSig : REFERENCE TO BOOL;
	p_bAOIOriginSig : REFERENCE TO BOOL;
	p_bBuzAlertEn : REFERENCE TO BOOL;
	p_bTLBlueFlashEn : REFERENCE TO BOOL;
	p_bTLAmberFlashEn : REFERENCE TO BOOL;
	p_bTLWhiteFlashEn : REFERENCE TO BOOL;
	p_bTLRedFlashEn : REFERENCE TO BOOL;
	p_bTLGreenFlashEn : REFERENCE TO BOOL;
END_VAR
(*Add*)
VAR
	p_tyBuffer1BffrStat : REFERENCE TO tyBffrStat;
	p_tyBuffer2BffrStat : REFERENCE TO tyBffrStat;
	p_tyBuffer3BffrStat : REFERENCE TO tyBffrStat;
	p_bMcParamAGVComEn : REFERENCE TO BOOL;
	p_eMcParamMagExMode : REFERENCE TO eMcMagExchangeMode;
END_VAR
```

#### InputRef_Link.var
```iecst
(*2019-04-09*)
VAR
	p_bLinkAlarmWarning : REFERENCE TO BOOL;
	p_bLinkAlarmInfo : REFERENCE TO BOOL;
	p_bLinkUIWarning : REFERENCE TO BOOL;
	p_bLinkAlarmInfoLF : REFERENCE TO BOOL;
	p_bLinkLFBuzMute : REFERENCE TO BOOL;
	p_bLinkMagFullTLMuteBuzz : REFERENCE TO BOOL;
	p_bLinkMagFullInfo : REFERENCE TO BOOL;
END_VAR
(**)
(*MEK*)
VAR
	p_bLinkAOIOrgOK1 : REFERENCE TO BOOL;
	p_bLinkAOIOrgOK2 : REFERENCE TO BOOL;
	p_bLinkAOIErr1 : REFERENCE TO BOOL;
	p_bLinkAOIErr2 : REFERENCE TO BOOL;
	p_usiLinkMcMod : REFERENCE TO USINT;
END_VAR
(**)
(*BHTC*)
VAR
	p_bLinkMagazineEmpty : REFERENCE TO BOOL;
	p_bLinkUpperMagazineFull : REFERENCE TO BOOL;
	p_bLinkLowerMagazineEmpty : REFERENCE TO BOOL;
	p_bLinkStackEmpty : REFERENCE TO BOOL;
	p_bLinkStackAlmostEmpty : REFERENCE TO BOOL;
	p_bLinkSPIBadPCB : REFERENCE TO BOOL;
	p_bLinkRescanning : REFERENCE TO BOOL;
	p_bLinkRescanFail : REFERENCE TO BOOL;
	p_bLinkBadRejected : REFERENCE TO BOOL;
	p_bLinkBadRejectedwithUBAB : REFERENCE TO BOOL;
	p_bLinkCounterUp : REFERENCE TO BOOL;
	p_bLinkCounterUpNHalf : REFERENCE TO BOOL;
	p_bLinkOvenInfoReceived : REFERENCE TO BOOL;
	p_bLinkThresholdSignal : REFERENCE TO BOOL;
	p_bLinkTwoPCBRejected : REFERENCE TO BOOL;
	p_bLinkUpperMagazineEmpty : REFERENCE TO BOOL;
	p_bLinkLowerMagazineFull : REFERENCE TO BOOL;
END_VAR
(**)
```

#### Local.var
```iecst
(*2020-03-16*)
(**)
(*Local Action, State & Status*)
VAR
	eAct : eTLBuzAction := TLBuzActIdle;
	eStat : eTLBuzAction := TLBuzActIdle;
	eStatus : eFBStatus := Idle;
	sStatTxt : STRING[200] := '';
	a_sStatText : ARRAY[0..50] OF STRING[200] := ['Idling','Turning On Tower Light Green','Turning On Tower Light Amber','Turning On Tower Light Red','Turning On Buzzer','Turning Off Tower Light Green','Turning Off Tower Light Amber','Turning Off Tower Light Red','Turning Off Buzzer','Turning On All Output','Turning Off All Output',40('')];
END_VAR
(**)
(*Local Alarm*)
(**)
(*Local Output*)
VAR
	bTLBlue : BOOL;
	bTLRed : BOOL;
	bTLAmber : BOOL;
	bTLWhite : BOOL;
	bTLGreen : BOOL;
	bBuzBeep : BOOL;
END_VAR
(**)
(*Local Input*)
VAR
	bManualErrOn : BOOL := FALSE;
	bManual : BOOL := FALSE;
	bStartup : BOOL := FALSE;
	bErr : BOOL := FALSE;
	bErrNoBuz : BOOL := FALSE;
	bWarning : BOOL := FALSE;
	bWarningNoBuz : BOOL := FALSE;
	bWarning1 : BOOL := FALSE;
	bWarning1NoBuz : BOOL := FALSE;
	bWarning2 : BOOL := FALSE;
	bWarning2NoBuz : BOOL := FALSE;
	bWarning3 : BOOL := FALSE;
	bWarning3NoBuz : BOOL := FALSE;
	bWarning4 : BOOL := FALSE;
	bWarning4NoBuz : BOOL := FALSE;
	bWarning5 : BOOL := FALSE;
	bWarning5NoBuz : BOOL := FALSE;
	bChgRcp : BOOL := FALSE;
	bSeqStop : BOOL := FALSE;
	bStep : BOOL := FALSE;
	bOps : BOOL := FALSE;
	bStandby : BOOL := FALSE;
	bSimulation : BOOL := FALSE;
	bMuteBuz : BOOL := FALSE;
	tTLChgRcpBlinkTm : TIME := T#200ms;
	tTLErrBlinkTm : TIME := T#500ms;
	tBuzErrOnTm : TIME := T#500ms;
	tBuzErrRestTm : TIME := T#500ms;
	usiBuzErrOnCntr : USINT := 3;
	bBuzErrStopSeqEn : BOOL := FALSE;
	usiBuzErrStopSeqCntr : USINT := 3;
	tTLWarnBlinkTm : TIME := T#500ms;
	tBuzWarnOnTm : TIME := T#500ms;
	tBuzWarnRestTm : TIME := T#5s;
	usiBuzWarnOnCntr : USINT := 3;
	bBuzWarnStopSeqEn : BOOL := FALSE;
	usiBuzWarnStopSeqCntr : USINT := 3;
	tTLWarn1BlinkTm : TIME := T#500ms;
	tBuzWarn1OnTm : TIME := T#500ms;
	tBuzWarn1RestTm : TIME := T#5s;
	usiBuzWarn1OnCntr : USINT := 3;
	bBuzWarn1StopSeqEn : BOOL := FALSE;
	usiBuzWarn1StopSeqCntr : USINT := 3;
	tTLWarn2BlinkTm : TIME := T#500ms;
	tBuzWarn2OnTm : TIME := T#500ms;
	tBuzWarn2RestTm : TIME := T#5s;
	usiBuzWarn2OnCntr : USINT := 3;
	bBuzWarn2StopSeqEn : BOOL := FALSE;
	usiBuzWarn2StopSeqCntr : USINT := 3;
	tTLWarn3BlinkTm : TIME := T#500ms;
	tBuzWarn3OnTm : TIME := T#500ms;
	tBuzWarn3RestTm : TIME := T#5s;
	usiBuzWarn3OnCntr : USINT := 3;
	bBuzWarn3StopSeqEn : BOOL := FALSE;
	usiBuzWarn3StopSeqCntr : USINT := 3;
	tTLWarn4BlinkTm : TIME := T#500ms;
	tBuzWarn4OnTm : TIME := T#500ms;
	tBuzWarn4RestTm : TIME := T#5s;
	usiBuzWarn4OnCntr : USINT := 3;
	bBuzWarn4StopSeqEn : BOOL := FALSE;
	usiBuzWarn4StopSeqCntr : USINT := 3;
	tTLWarn5BlinkTm : TIME := T#500ms;
	tBuzWarn5OnTm : TIME := T#500ms;
	tBuzWarn5RestTm : TIME := T#5s;
	usiBuzWarn5OnCntr : USINT := 3;
	bBuzWarn5StopSeqEn : BOOL := FALSE;
	usiBuzWarn5StopSeqCntr : USINT := 3;
	tBuzAlertOnTm : TIME := T#500ms;
	tBuzAlertRestTm : TIME := T#5s;
	usiBuzAlertOnCntr : USINT := 3;
	bBuzAlertStopSeqEn : BOOL := FALSE;
	usiBuzAlertStopSeqCntr : USINT := 3;
	tTLBlueBlinkTm : TIME := T#500ms;
	tTLAmberBlinkTm : TIME := T#500ms;
	tTLWhiteBlinkTm : TIME := T#500ms;
	tTLRedBlinkTm : TIME := T#500ms;
	tTLGreenBlinkTm : TIME := T#500ms;
	bCoveSwitchSig : BOOL := FALSE;
	eTLBuzMode : eTLBuzMod := TLBuzModNutek;
	bAOIErrSig : BOOL := FALSE;
	bAOIOriginSig : BOOL := FALSE;
	bBuzAlertEn : BOOL := FALSE;
	bTLBlueFlashEn : BOOL := FALSE;
	bTLAmberFlashEn : BOOL := FALSE;
	bTLWhiteFlashEn : BOOL := FALSE;
	bTLRedFlashEn : BOOL := FALSE;
	bTLGreenFlashEn : BOOL := FALSE;
END_VAR
(**)
(*Local*)
VAR
	usiWarnInfoStateOld : USINT; (*Default buzzer behavior*)
	usiWarnInfoStateNew : USINT; (*Default buzzer behavior*)
	bInitDone : BOOL;
	bInitialDone : BOOL;
	tBlinkTm : TIME := T#500ms;
	fbBlink : fbTLBuzBlink;
	fbBlink1 : fbTLBuzBlink;
	fbBlink2 : fbTLBuzBlink;
	fbBlink3 : fbTLBuzBlink;
	fbBlink4 : fbTLBuzBlink;
	fbWarning : fbTLBuzWarn;
	fbWarning1 : fbTLBuzWarn;
	eStatOld : eTLBuzAction := TLBuzActIdle;
	bEmptyMag : BOOL := FALSE;
END_VAR
```

#### Act_Background.st
```iecst
(** 2020-10-05 **)
ACTION Act_Background: //For Standard Machines

	IF EDGEPOS(p_bManual) THEN

		fbBlink(bEn := FALSE);
		fbWarning(bEn := FALSE);

		bTLRed		:= FALSE;
		bTLAmber	:= TRUE;
		bTLGreen	:= FALSE;
		bBuzBeep	:= FALSE;

	ELSIF p_bManual THEN

		IF p_bErr = TRUE THEN

			fbBlink.tOnTm	:= p_tTLErrBlinkTm; //Error T#500ms (from NtParam)
			fbBlink.tOffTm	:= p_tTLErrBlinkTm; //Error T#500ms (from NtParam)

			fbWarning.tOnTm					:= p_tBuzErrOnTm; //Warn T#500ms (from NtParam)
			fbWarning.tOffTm				:= p_tBuzErrOnTm; //Warn T#500ms (from NtParam)
			fbWarning.tRstTm				:= p_tBuzErrRestTm; //Rest 5 seconds (from NtParam)
			fbWarning.usiOnCnt				:= p_usiBuzErrOnCntr; //Count 3 times (from NtParam)
			fbWarning.bStopAftRptSeqEn		:= p_bBuzErrStopSeqEn; //Enable Sequence Count (from NtParam)
			fbWarning.usiStopAftRptSeqCntr	:= p_usiBuzErrStopSeqCntr; //Sequence Counter  (from NtParam)

			fbBlink(bEn := TRUE);
			fbWarning(bEn := TRUE);

			bTLRed		:= fbBlink.bOut;
			bBuzBeep	:= (fbWarning.bOut) AND (p_bMuteBuz = FALSE);

			bManualErrOn := TRUE;

		ELSIF bManualErrOn THEN

			fbBlink(bEn := FALSE);
			fbWarning(bEn := FALSE);

			bTLRed		:= FALSE;
			bBuzBeep	:= FALSE;

			bManualErrOn := FALSE;

		END_IF

	ELSIF p_bManual = FALSE THEN

		bManualErrOn := FALSE;

		IF p_bStartup = TRUE THEN

			fbBlink(bEn := FALSE);
			fbWarning(bEn := FALSE);

			bTLRed		:= TRUE;
			bTLAmber	:= TRUE;
			bTLGreen	:= TRUE;
			bBuzBeep	:= FALSE;

		ELSIF p_bErr = TRUE THEN

			fbBlink.tOnTm	:= p_tTLErrBlinkTm; //Error T#500ms (from NtParam)
			fbBlink.tOffTm	:= p_tTLErrBlinkTm; //Error T#500ms (from NtParam)

			fbWarning.tOnTm					:= p_tBuzErrOnTm; //Warn T#500ms (from NtParam)
			fbWarning.tOffTm				:= p_tBuzErrOnTm; //Warn T#500ms (from NtParam)
			fbWarning.tRstTm				:= p_tBuzErrRestTm; //Rest 5 seconds (from NtParam)
			fbWarning.usiOnCnt				:= p_usiBuzErrOnCntr; //Count 3 times (from NtParam)
			fbWarning.bStopAftRptSeqEn		:= p_bBuzErrStopSeqEn; //Enable Sequence Count (from NtParam)
			fbWarning.usiStopAftRptSeqCntr	:= p_usiBuzErrStopSeqCntr; //Sequence Counter  (from NtParam)

			fbBlink(bEn := TRUE);
			fbWarning(bEn := TRUE);

			bTLRed		:= fbBlink.bOut;
			bTLAmber	:= FALSE;
			bTLGreen	:= FALSE;
			bBuzBeep	:= (fbWarning.bOut) AND (p_bMuteBuz = FALSE);

		ELSIF p_bErrNoBuz = TRUE THEN

			fbBlink.tOnTm	:= p_tTLErrBlinkTm;
			fbBlink.tOffTm	:= p_tTLErrBlinkTm;
			fbBlink(bEn := TRUE);
			fbWarning(bEn := FALSE);

			bTLRed		:= fbBlink.bOut;
			bTLAmber	:= FALSE;
			bTLGreen	:= FALSE;
			bBuzBeep	:= FALSE;

		ELSIF p_bWarning = TRUE THEN

			fbBlink.tOnTm	:= p_tTLWarnBlinkTm; //Warn T#500ms (from NtParam)
			fbBlink.tOffTm	:= p_tTLWarnBlinkTm; //Warn T#500ms (from NtParam)

			fbWarning.tOnTm					:= p_tBuzWarnOnTm; //Warn T#500ms (from NtParam)
			fbWarning.tOffTm				:= p_tBuzWarnOnTm; //Warn T#500ms (from NtParam)
			fbWarning.tRstTm				:= p_tBuzWarnRestTm; //Rest 5 seconds (from NtParam)
			fbWarning.usiOnCnt				:= p_usiBuzWarnOnCntr; //Count 3 times (from NtParam)
			fbWarning.bStopAftRptSeqEn		:= p_bBuzWarnStopSeqEn; //Enable Sequence Count (from NtParam)
			fbWarning.usiStopAftRptSeqCntr	:= p_usiBuzWarnStopSeqCntr; //Sequence Counter  (from NtParam)

			fbBlink(bEn := TRUE);
			fbWarning(bEn := TRUE);

			bTLRed		:= p_bStandby;
			bTLAmber	:= fbBlink.bOut;
			bTLGreen	:= p_bOps;
			bBuzBeep	:= fbWarning.bOut AND (p_bMuteBuz = FALSE);

		ELSIF p_bWarningNoBuz = TRUE THEN

			fbBlink.tOnTm	:= p_tTLWarnBlinkTm;
			fbBlink.tOffTm	:= p_tTLWarnBlinkTm;
			fbBlink(bEn := TRUE);
			fbWarning(bEn := FALSE);

			bTLRed		:= p_bStandby;
			bTLAmber	:= fbBlink.bOut;
			bTLGreen	:= p_bOps;
			bBuzBeep	:= FALSE;

		ELSIF p_bWarning1 = TRUE THEN

			fbBlink.tOnTm	:= p_tTLWarn1BlinkTm;
			fbBlink.tOffTm	:= p_tTLWarn1BlinkTm;

			fbWarning.tOnTm					:= p_tBuzWarn1OnTm; //Warn T#500ms (from NtParam)
			fbWarning.tOffTm				:= p_tBuzWarn1OnTm; //Warn T#500ms (from NtParam)
			fbWarning.tRstTm				:= p_tBuzWarn1RestTm; //Rest 5 seconds (from NtParam)
			fbWarning.usiOnCnt				:= p_usiBuzWarn1OnCntr; //Count 3 times (from NtParam)
			fbWarning.bStopAftRptSeqEn		:= p_bBuzWarn1StopSeqEn; //Enable Sequence Count (from NtParam)
			fbWarning.usiStopAftRptSeqCntr	:= p_usiBuzWarn1StopSeqCntr; //Sequence Counter  (from NtParam)

			fbBlink(bEn := TRUE);
			fbWarning(bEn := TRUE);

			bTLRed		:= p_bStandby;
			bTLAmber	:= fbBlink.bOut;
			bTLGreen	:= p_bOps;
			bBuzBeep	:= fbWarning.bOut AND (p_bMuteBuz = FALSE);

		ELSIF p_bWarning1NoBuz = TRUE THEN

			fbBlink.tOnTm	:= p_tTLWarn1BlinkTm;
			fbBlink.tOffTm	:= p_tTLWarn1BlinkTm;
			fbBlink(bEn := TRUE);
			fbWarning(bEn := FALSE);

			bTLRed		:= p_bStandby;
			bTLAmber	:= fbBlink.bOut;
			bTLGreen	:= p_bOps;
			bBuzBeep	:= FALSE;

		ELSIF p_bWarning2 = TRUE THEN

			fbBlink.tOnTm	:= p_tTLWarn2BlinkTm;
			fbBlink.tOffTm	:= p_tTLWarn2BlinkTm;

			fbWarning.tOnTm					:= p_tBuzWarn2OnTm; //Warn T#500ms (from NtParam)
			fbWarning.tOffTm				:= p_tBuzWarn2OnTm; //Warn T#500ms (from NtParam)
			fbWarning.tRstTm				:= p_tBuzWarn2RestTm; //Rest 5 seconds (from NtParam)
			fbWarning.usiOnCnt				:= p_usiBuzWarn2OnCntr; //Count 3 times (from NtParam)
			fbWarning.bStopAftRptSeqEn		:= p_bBuzWarn2StopSeqEn; //Enable Sequence Count (from NtParam)
			fbWarning.usiStopAftRptSeqCntr	:= p_usiBuzWarn2StopSeqCntr; //Sequence Counter  (from NtParam)

			fbBlink(bEn := TRUE);
			fbWarning(bEn := TRUE);

			bTLRed		:= p_bStandby;
			bTLAmber	:= fbBlink.bOut;
			bTLGreen	:= p_bOps;
			bBuzBeep	:= fbWarning.bOut AND (p_bMuteBuz = FALSE);

		ELSIF p_bWarning2NoBuz = TRUE THEN

			fbBlink.tOnTm	:= p_tTLWarn2BlinkTm;
			fbBlink.tOffTm	:= p_tTLWarn2BlinkTm;
			fbBlink(bEn := TRUE);
			fbWarning(bEn := FALSE);

			bTLRed		:= p_bStandby;
			bTLAmber	:= fbBlink.bOut;
			bTLGreen	:= p_bOps;
			bBuzBeep	:= FALSE;

		ELSIF p_bWarning3 = TRUE THEN

			fbBlink.tOnTm	:= p_tTLWarn3BlinkTm;
			fbBlink.tOffTm	:= p_tTLWarn3BlinkTm;

			fbWarning.tOnTm					:= p_tBuzWarn3OnTm; //Warn T#500ms (from NtParam)
			fbWarning.tOffTm				:= p_tBuzWarn3OnTm; //Warn T#500ms (from NtParam)
			fbWarning.tRstTm				:= p_tBuzWarn3RestTm; //Rest 5 seconds (from NtParam)
			fbWarning.usiOnCnt				:= p_usiBuzWarn3OnCntr; //Count 3 times (from NtParam)
			fbWarning.bStopAftRptSeqEn		:= p_bBuzWarn3StopSeqEn; //Enable Sequence Count (from NtParam)
			fbWarning.usiStopAftRptSeqCntr	:= p_usiBuzWarn3StopSeqCntr; //Sequence Counter  (from NtParam)

			fbBlink(bEn := TRUE);
			fbWarning(bEn := TRUE);

			bTLRed		:= p_bStandby;
			bTLAmber	:= fbBlink.bOut;
			bTLGreen	:= p_bOps;
			bBuzBeep	:= fbWarning.bOut AND (p_bMuteBuz = FALSE);

		ELSIF p_bWarning3NoBuz = TRUE THEN

			fbBlink.tOnTm	:= p_tTLWarn3BlinkTm;
			fbBlink.tOffTm	:= p_tTLWarn3BlinkTm;
			fbBlink(bEn := TRUE);
			fbWarning(bEn := FALSE);

			bTLRed		:= p_bStandby;
			bTLAmber	:= fbBlink.bOut;
			bTLGreen	:= p_bOps;
			bBuzBeep	:= FALSE;

		ELSIF p_bWarning4 = TRUE THEN

			fbBlink.tOnTm	:= p_tTLWarn4BlinkTm;
			fbBlink.tOffTm	:= p_tTLWarn4BlinkTm;

			fbWarning.tOnTm					:= p_tBuzWarn4OnTm; //Warn T#500ms (from NtParam)
			fbWarning.tOffTm				:= p_tBuzWarn4OnTm; //Warn T#500ms (from NtParam)
			fbWarning.tRstTm				:= p_tBuzWarn4RestTm; //Rest 5 seconds (from NtParam)
			fbWarning.usiOnCnt				:= p_usiBuzWarn4OnCntr; //Count 3 times (from NtParam)
			fbWarning.bStopAftRptSeqEn		:= p_bBuzWarn4StopSeqEn; //Enable Sequence Count (from NtParam)
			fbWarning.usiStopAftRptSeqCntr	:= p_usiBuzWarn4StopSeqCntr; //Sequence Counter  (from NtParam)

			fbBlink(bEn := TRUE);
			fbWarning(bEn := TRUE);

			bTLRed		:= p_bStandby;
			bTLAmber	:= fbBlink.bOut;
			bTLGreen	:= p_bOps;
			bBuzBeep	:= fbWarning.bOut AND (p_bMuteBuz = FALSE);

		ELSIF p_bWarning4NoBuz = TRUE THEN

			fbBlink.tOnTm	:= p_tTLWarn4BlinkTm;
			fbBlink.tOffTm	:= p_tTLWarn4BlinkTm;
			fbBlink(bEn := TRUE);
			fbWarning(bEn := FALSE);

			bTLRed		:= p_bStandby;
			bTLAmber	:= fbBlink.bOut;
			bTLGreen	:= p_bOps;
			bBuzBeep	:= FALSE;

		ELSIF p_bWarning5 = TRUE THEN

			fbBlink.tOnTm	:= p_tTLWarn5BlinkTm;
			fbBlink.tOffTm	:= p_tTLWarn5BlinkTm;

			fbWarning.tOnTm					:= p_tBuzWarn5OnTm; //Warn T#500ms (from NtParam)
			fbWarning.tOffTm				:= p_tBuzWarn5OnTm; //Warn T#500ms (from NtParam)
			fbWarning.tRstTm				:= p_tBuzWarn5RestTm; //Rest 5 seconds (from NtParam)
			fbWarning.usiOnCnt				:= p_usiBuzWarn5OnCntr; //Count 3 times (from NtParam)
			fbWarning.bStopAftRptSeqEn		:= p_bBuzWarn5StopSeqEn; //Enable Sequence Count (from NtParam)
			fbWarning.usiStopAftRptSeqCntr	:= p_usiBuzWarn5StopSeqCntr; //Sequence Counter  (from NtParam)

			fbBlink(bEn := TRUE);
			fbWarning(bEn := TRUE);

			bTLRed		:= p_bStandby;
			bTLAmber	:= fbBlink.bOut;
			bTLGreen	:= p_bOps;
			bBuzBeep	:= fbWarning.bOut AND (p_bMuteBuz = FALSE);

		ELSIF p_bWarning5NoBuz = TRUE THEN

			fbBlink.tOnTm	:= p_tTLWarn5BlinkTm;
			fbBlink.tOffTm	:= p_tTLWarn5BlinkTm;
			fbBlink(bEn := TRUE);
			fbWarning(bEn := FALSE);

			bTLRed		:= p_bStandby;
			bTLAmber	:= fbBlink.bOut;
			bTLGreen	:= p_bOps;
			bBuzBeep	:= FALSE;

		ELSIF p_bSeqStop = TRUE THEN

			fbBlink.tOnTm	:= tBlinkTm;
			fbBlink.tOffTm	:= tBlinkTm;
			fbBlink(bEn := TRUE);
			fbWarning(bEn := FALSE);

			bTLRed		:= fbBlink.bOut;
			bTLAmber	:= FALSE;
			bTLGreen	:= TRUE;
			bBuzBeep	:= FALSE;

		ELSIF p_bChgRcp = TRUE THEN

			fbBlink.tOnTm	:= p_tTLChgRcpBlinkTm;
			fbBlink.tOffTm	:= p_tTLChgRcpBlinkTm;
			fbBlink(bEn := TRUE);
			fbWarning(bEn := FALSE);

			IF EDGE(fbBlink.bOut) THEN
				IF bTLRed = TRUE THEN
					bTLRed		:= FALSE;
					bTLAmber	:= FALSE;
					bTLGreen	:= TRUE;
				ELSIF bTLAmber = TRUE THEN
					bTLRed		:= TRUE;
					bTLAmber	:= FALSE;
					bTLGreen	:= FALSE;
				ELSE
					bTLRed		:= FALSE;
					bTLAmber	:= TRUE;
					bTLGreen	:= FALSE;
				END_IF
			END_IF

			bBuzBeep	:= fbBlink.bOut AND (p_bMuteBuz = FALSE);

		ELSIF p_bStep = TRUE THEN

			fbBlink.tOnTm	:= tBlinkTm;
			fbBlink.tOffTm	:= tBlinkTm;
			fbBlink(bEn := TRUE);
			fbWarning(bEn := FALSE);

			bTLRed		:= FALSE;
			bTLAmber	:= FALSE;
			bTLGreen	:= fbBlink.bOut;
			bBuzBeep	:= FALSE;

		ELSIF p_bOps = TRUE THEN

			fbBlink(bEn := FALSE);
			fbWarning(bEn := FALSE);

			bTLRed		:= FALSE;
			bTLAmber	:= FALSE;
			bTLGreen	:= TRUE;
			bBuzBeep	:= FALSE;

		ELSIF p_bSimulation = TRUE THEN

			fbBlink.tOnTm	:= tBlinkTm;
			fbBlink.tOffTm	:= tBlinkTm;
			fbBlink(bEn := TRUE);
			fbWarning(bEn := FALSE);

			bTLRed		:= fbBlink.bOut;
			bTLAmber	:= fbBlink.bOut;
			bTLGreen	:= TRUE;
			bBuzBeep	:= FALSE;

		ELSIF p_bStandby = TRUE THEN

			fbBlink(bEn := FALSE);
			fbWarning(bEn := FALSE);

			bTLRed		:= TRUE;
			bTLAmber	:= FALSE;
			bTLGreen	:= FALSE;
			bBuzBeep	:= FALSE;

		ELSE

			fbBlink(bEn := FALSE);
			fbWarning(bEn := FALSE);

			bTLRed		:= FALSE;
			bTLAmber	:= FALSE;
			bTLGreen	:= FALSE;
			bBuzBeep	:= FALSE;

		END_IF

	END_IF

	IF p_bManual = FALSE AND p_bErr = FALSE THEN
		IF p_bTLAmberFlashEn THEN //Amber Flash 1 sec [Put Conditions in Act_Link.st]

			fbBlink1.tOnTm	:= p_tTLAmberBlinkTm; //T#500ms (from NtParam)
			fbBlink1.tOffTm	:= p_tTLAmberBlinkTm; //T#500ms (from NtParam)
			fbBlink1(bEn := TRUE);

			bTLAmber	:= fbBlink1.bOut;

		ELSE
			fbBlink1(bEn := FALSE);
		END_IF

		IF p_bTLRedFlashEn THEN //Red Flash 1 sec [Put Conditions in Act_Link.st]

			fbBlink2.tOnTm	:= p_tTLRedBlinkTm; //T#500ms (from NtParam)
			fbBlink2.tOffTm	:= p_tTLRedBlinkTm; //T#500ms (from NtParam)
			fbBlink2(bEn := TRUE);

			bTLRed		:= fbBlink2.bOut;
		ELSE
			fbBlink2(bEn := FALSE);
		END_IF

		IF p_bTLGreenFlashEn THEN //Green Flash 1 sec [Put Conditions in Act_Link.st]

			fbBlink3.tOnTm	:= p_tTLGreenBlinkTm; //T#500ms (from NtParam)
			fbBlink3.tOffTm	:= p_tTLGreenBlinkTm; //T#500ms (from NtParam)
			fbBlink3(bEn := TRUE);

			bTLGreen	:= fbBlink3.bOut;
		ELSE
			fbBlink3(bEn := FALSE);
		END_IF

		IF p_bBuzAlertEn = TRUE AND fbWarning.bEn=FALSE THEN

			fbWarning1.tOnTm				:= p_tBuzAlertOnTm;
			fbWarning1.tOffTm				:= p_tBuzAlertOnTm;
			fbWarning1.tRstTm				:= p_tBuzAlertRestTm;
			fbWarning1.usiOnCnt				:= p_usiBuzAlertOnCntr;
			fbWarning1.bStopAftRptSeqEn		:= p_bBuzAlertStopSeqEn; //Enable Sequence Count (from NtParam)
			fbWarning1.usiStopAftRptSeqCntr	:= p_usiBuzAlertStopSeqCntr; //Sequence Counter  (from NtParam)

			fbWarning1(bEn := TRUE);

			bBuzBeep	:= fbWarning1.bOut AND (p_bMuteBuz = FALSE);

		ELSE
			fbWarning1(bEn := FALSE);
		END_IF
	ELSE
		fbBlink1(bEn := FALSE);
		fbBlink2(bEn := FALSE);
		fbBlink3(bEn := FALSE);
		fbWarning1(bEn := FALSE);
	END_IF

	//Arrange p_bWarning according to the severity of the warning or info (Err is prioritized)
	IF p_bErr THEN
		usiWarnInfoStateNew	:= 1;
	ELSIF p_bWarning THEN
		usiWarnInfoStateNew	:= 2;
	ELSIF p_bWarning1 THEN
		usiWarnInfoStateNew	:= 3;
	ELSIF p_bWarning2 THEN
		usiWarnInfoStateNew	:= 4;
	ELSIF p_bWarning3 THEN
		usiWarnInfoStateNew	:= 5;
	ELSIF p_bWarning4 THEN
		usiWarnInfoStateNew	:= 6;
	ELSIF p_bWarning5 THEN
		usiWarnInfoStateNew	:= 7;
	ELSIF p_bBuzAlertEn AND fbWarning.bEn=FALSE THEN
		usiWarnInfoStateNew	:= 8;
	ELSE
		usiWarnInfoStateNew	:= 0;
	END_IF

	IF usiWarnInfoStateOld<>usiWarnInfoStateNew THEN
		usiWarnInfoStateOld:=usiWarnInfoStateNew;
		fbWarning(bEn := FALSE);
		fbWarning1(bEn := FALSE);
	END_IF

END_ACTION
```

#### Act_Background4.st
```iecst
ACTION Act_Background4:

	IF EDGEPOS(p_bManual) THEN

		fbBlink(bEn := FALSE);
		fbWarning(bEn := FALSE);

		bTLRed		:= FALSE;
		bTLAmber	:= TRUE;
		bTLGreen	:= FALSE;
		bBuzBeep	:= FALSE;
		bTLWhite	:= TRUE;

	ELSIF p_bManual THEN
//		bTLGreen := FALSE;
//		bTLWhite := TRUE;
//		bTLGreenFlashEn := FALSE;
//		bTLWhiteFlashEn := FALSE;
//		bBuzBeep := FALSE;
//		p_bBuzAlertEn := FALSE;

		IF p_bErr = TRUE THEN

			fbBlink.tOnTm	:= p_tTLErrBlinkTm; //Error T#500ms (from NtParam)
			fbBlink.tOffTm	:= p_tTLErrBlinkTm; //Error T#500ms (from NtParam)

			fbWarning.tOnTm					:= p_tBuzErrOnTm; //Warn T#500ms (from NtParam)
			fbWarning.tOffTm				:= p_tBuzErrOnTm; //Warn T#500ms (from NtParam)
			fbWarning.tRstTm				:= p_tBuzErrRestTm; //Rest 5 seconds (from NtParam)
			fbWarning.usiOnCnt				:= p_usiBuzErrOnCntr; //Count 3 times (from NtParam)
			fbWarning.bStopAftRptSeqEn		:= p_bBuzErrStopSeqEn; //Enable Sequence Count (from NtParam)
			fbWarning.usiStopAftRptSeqCntr	:= p_usiBuzErrStopSeqCntr; //Sequence Counter  (from NtParam)

			fbBlink(bEn := TRUE);
			fbWarning(bEn := TRUE);

			bTLRed		:= fbBlink.bOut;
			bBuzBeep	:= (fbWarning.bOut) AND (p_bMuteBuz = FALSE);

			bManualErrOn := TRUE;
			p_bBuzAlertEn := FALSE;

		ELSIF bManualErrOn THEN

			fbBlink(bEn := FALSE);
			fbWarning(bEn := FALSE);

			bTLRed		:= FALSE;
			bBuzBeep	:= FALSE;

			bManualErrOn := FALSE;
			p_bBuzAlertEn := FALSE;

		END_IF

	ELSIF p_bManual = FALSE THEN

		bManualErrOn := FALSE;

		IF p_bStartup THEN
			bTLGreen := FALSE;
			bTLWhite := FALSE;
			bTLGreenFlashEn := TRUE;
			bTLWhiteFlashEn := TRUE;
			bBuzBeep := FALSE;
			p_bBuzAlertEn := FALSE;

		ELSIF p_bOps THEN
			bTLGreen := TRUE;
			bTLWhite := FALSE;
			bTLGreenFlashEn := FALSE;
			bTLWhiteFlashEn := FALSE;
			bBuzBeep := FALSE;
			p_bBuzAlertEn := FALSE;

		ELSIF p_bSeqStop THEN
			bTLGreen := FALSE;
			bTLWhite := FALSE;
			bTLGreenFlashEn := TRUE;
			bTLWhiteFlashEn := FALSE;
			bBuzBeep := FALSE;
			p_bBuzAlertEn := FALSE;

		ELSIF p_bStandby THEN
			bTLGreen := FALSE;
			bTLWhite := FALSE;
			bTLGreenFlashEn := FALSE;
			bTLWhiteFlashEn := TRUE;
			bBuzBeep := FALSE;
			p_bBuzAlertEn := FALSE;

		ELSIF p_bSimulation THEN
			bTLGreen := TRUE;
			bTLWhite := FALSE;
			bTLGreenFlashEn := FALSE;
			bTLWhiteFlashEn := TRUE;
			bBuzBeep := FALSE;
			p_bBuzAlertEn := FALSE;

		END_IF

		bEmptyMag :=(p_tyBuffer1BffrStat.bBffrMty OR p_tyBuffer2BffrStat.bBffrMty OR p_tyBuffer3BffrStat.bBffrMty);

		IF p_bMcParamAGVComEn THEN
			IF bEmptyMag THEN
				IF p_bOps THEN
					bTLGreen := TRUE;
				ELSE
					bTLGreen := FALSE;
				END_IF
				bTLWhite := FALSE;
				bTLGreenFlashEn := FALSE;
				bTLWhiteFlashEn := TRUE;
				bBuzBeep := FALSE;
				p_bBuzAlertEn := FALSE;
			END_IF
		END_IF

		IF p_bWarning THEN
			IF p_bOps THEN
				bTLGreen := TRUE;
				bTLWhite := FALSE;
				bTLGreenFlashEn := FALSE;
				bTLWhiteFlashEn := TRUE;
			ELSIF p_bSeqStop THEN
				bTLGreen := FALSE;
				bTLWhite := FALSE;
				bTLGreenFlashEn := TRUE;
				bTLWhiteFlashEn := TRUE;
			ELSE
				bTLGreen := FALSE;
				bTLWhite := FALSE;
				bTLGreenFlashEn := FALSE;
				bTLWhiteFlashEn := TRUE;
			END_IF

			IF p_eMcParamMagExMode =  McSetMagXcAutoMode THEN
				p_bBuzAlertEn := FALSE;
			ELSE
				p_bBuzAlertEn := TRUE;
			END_IF

//			IF bBuzBeep AND p_bMcParamAGVComEn AND bEmptyMag THEN
//				bBuzBeep := FALSE;
//			ELSE
//				bBuzBeep := TRUE;
//			END_IF
//			p_bBuzAlertEn := TRUE;
		END_IF

		IF p_bErr THEN
			fbBlink.tOnTm	:= p_tTLErrBlinkTm; //Error T#500ms (from NtParam)
			fbBlink.tOffTm	:= p_tTLErrBlinkTm; //Error T#500ms (from NtParam)

			fbWarning.tOnTm					:= p_tBuzErrOnTm; //Warn T#500ms (from NtParam)
			fbWarning.tOffTm				:= p_tBuzErrOnTm; //Warn T#500ms (from NtParam)
			fbWarning.tRstTm				:= p_tBuzErrRestTm; //Rest 5 seconds (from NtParam)
			fbWarning.usiOnCnt				:= p_usiBuzErrOnCntr; //Count 3 times (from NtParam)
			fbWarning.bStopAftRptSeqEn		:= p_bBuzErrStopSeqEn; //Enable Sequence Count (from NtParam)
			fbWarning.usiStopAftRptSeqCntr	:= p_usiBuzErrStopSeqCntr; //Sequence Counter  (from NtParam)

			fbBlink(bEn := TRUE);
			fbWarning(bEn := TRUE);

			bTLRed		:= fbBlink.bOut;
			bTLAmber	:= FALSE;
			bTLGreen	:= FALSE;
			bBuzBeep	:= (fbWarning.bOut) AND (p_bMuteBuz = FALSE);
			p_bBuzAlertEn := FALSE;
		END_IF

		IF bTLWhiteFlashEn THEN //White Flash 1 sec [Put Conditions in Act_Link.st]

			fbBlink2.tOnTm	:= p_tTLWhiteBlinkTm; //T#500ms (from NtParam)
			fbBlink2.tOffTm	:= p_tTLWhiteBlinkTm; //T#500ms (from NtParam)
			fbBlink2(bEn := TRUE);

			bTLWhite		:= fbBlink2.bOut;
		ELSE
			fbBlink2(bEn := FALSE);
		END_IF

		IF bTLGreenFlashEn THEN //Green Flash 1 sec [Put Conditions in Act_Link.st]

			fbBlink3.tOnTm	:= p_tTLGreenBlinkTm; //T#500ms (from NtParam)
			fbBlink3.tOffTm	:= p_tTLGreenBlinkTm; //T#500ms (from NtParam)
			fbBlink3(bEn := TRUE);

			bTLGreen	:= fbBlink3.bOut;
		ELSE
			fbBlink3(bEn := FALSE);
		END_IF

		IF p_bBuzAlertEn THEN

			fbWarning1.tOnTm				:= p_tBuzAlertOnTm;
			fbWarning1.tOffTm				:= p_tBuzAlertOnTm;
			fbWarning1.tRstTm				:= p_tBuzAlertRestTm;
			fbWarning1.usiOnCnt				:= p_usiBuzAlertOnCntr;
			fbWarning1.bStopAftRptSeqEn		:= p_bBuzAlertStopSeqEn; //Enable Sequence Count (from NtParam)
			fbWarning1.usiStopAftRptSeqCntr	:= p_usiBuzAlertStopSeqCntr; //Sequence Counter  (from NtParam)

			fbWarning1(bEn := TRUE);

			bBuzBeep	:= fbWarning1.bOut AND (p_bMuteBuz = FALSE);

		ELSE
			fbWarning1(bEn := FALSE);
		END_IF
	END_IF

END_ACTION
```

#### Act_InitGlobal.st
```iecst
(** 2019-05-20 **)
ACTION Act_InitGlobal:

	//Pass Data To Link
	p_bLinkAlarmWarning ACCESS p_AlarmWarning;
	p_bLinkAlarmInfo ACCESS p_AlarmInfo;
	p_bLinkAlarmInfoLF ACCESS p_AlarmInfoLF;
	p_bLinkLFBuzMute ACCESS p_McParamLFBuzMute;

	//Pass Data To Internal Use
	p_bManual ACCESS p_UIUIMnlMod;
	p_bStartup ACCESS p_StartupRun;
	p_bErr ACCESS p_AlarmErr;
	p_bSeqStop ACCESS p_OpsStatusCycleStop;
	p_bStep ACCESS p_OpsStatusStep;
	p_bOps ACCESS p_OpsStatusRun;
	p_bStandby ACCESS p_OpsStatusStop;
	p_bMuteBuz ACCESS p_UIMuteBuz;
	p_bLinkMagFullTLMuteBuzz ACCESS p_OpsMagConvUL1TLMuteBuzz;
	p_bLinkMagFullInfo ACCESS p_OpsMagConvUL1MagFullInfo;

	//  -----------------------------------------  TLBuz 5.00.2  -----------------------------------------	//

	p_tTLChgRcpBlinkTm ACCESS p_NtParamTLChgRcpBlinkTm;

	p_tTLErrBlinkTm ACCESS p_NtParamTLErrBlinkTm;
	p_tBuzErrOnTm ACCESS p_NtParamBuzErrOnTm;
	p_tBuzErrRestTm ACCESS p_NtParamBuzErrRestTm;
	p_usiBuzErrOnCntr ACCESS p_NtParamBuzErrOnCntr;
	p_bBuzErrStopSeqEn ACCESS p_NtParamBuzErrStopSeqEn;
	p_usiBuzErrStopSeqCntr ACCESS p_NtParamBuzErrStopSeqCntr;

	p_tTLWarnBlinkTm ACCESS p_NtParamTLWarnBlinkTm;
	p_tBuzWarnOnTm ACCESS p_NtParamBuzWarnOnTm;
	p_tBuzWarnRestTm ACCESS p_NtParamBuzWarnRestTm;
	p_usiBuzWarnOnCntr ACCESS p_NtParamBuzWarnOnCntr;
	p_bBuzWarnStopSeqEn ACCESS p_NtParamBuzWarnStopSeqEn;
	p_usiBuzWarnStopSeqCntr ACCESS p_NtParamBuzWarnStopSeqCntr;

	p_tTLWarn1BlinkTm ACCESS p_NtParamTLWarn1BlinkTm;
	p_tBuzWarn1OnTm ACCESS p_NtParamBuzWarn1OnTm;
	p_tBuzWarn1RestTm ACCESS p_NtParamBuzWarn1RestTm;
	p_usiBuzWarn1OnCntr ACCESS p_NtParamBuzWarn1OnCntr;
	p_bBuzWarn1StopSeqEn ACCESS p_NtParamBuzWarn1StopSeqEn;
	p_usiBuzWarn1StopSeqCntr ACCESS p_NtParamBuzWarn1StopSeqCntr;

	p_tTLWarn2BlinkTm ACCESS p_NtParamTLWarn2BlinkTm;
	p_tBuzWarn2OnTm ACCESS p_NtParamBuzWarn2OnTm;
	p_tBuzWarn2RestTm ACCESS p_NtParamBuzWarn2RestTm;
	p_usiBuzWarn2OnCntr ACCESS p_NtParamBuzWarn2OnCntr;
	p_bBuzWarn2StopSeqEn ACCESS p_NtParamBuzWarn2StopSeqEn;
	p_usiBuzWarn2StopSeqCntr ACCESS p_NtParamBuzWarn2StopSeqCntr;

	p_tTLWarn3BlinkTm ACCESS p_NtParamTLWarn3BlinkTm;
	p_tBuzWarn3OnTm ACCESS p_NtParamBuzWarn3OnTm;
	p_tBuzWarn3RestTm ACCESS p_NtParamBuzWarn3RestTm;
	p_usiBuzWarn3OnCntr ACCESS p_NtParamBuzWarn3OnCntr;
	p_bBuzWarn3StopSeqEn ACCESS p_NtParamBuzWarn3StopSeqEn;
	p_usiBuzWarn3StopSeqCntr ACCESS p_NtParamBuzWarn3StopSeqCntr;

	p_tTLWarn4BlinkTm ACCESS p_NtParamTLWarn4BlinkTm;
	p_tBuzWarn4OnTm ACCESS p_NtParamBuzWarn4OnTm;
	p_tBuzWarn4RestTm ACCESS p_NtParamBuzWarn4RestTm;
	p_usiBuzWarn4OnCntr ACCESS p_NtParamBuzWarn4OnCntr;
	p_bBuzWarn4StopSeqEn ACCESS p_NtParamBuzWarn4StopSeqEn;
	p_usiBuzWarn4StopSeqCntr ACCESS p_NtParamBuzWarn4StopSeqCntr;

	p_tTLWarn5BlinkTm ACCESS p_NtParamTLWarn5BlinkTm;
	p_tBuzWarn5OnTm ACCESS p_NtParamBuzWarn5OnTm;
	p_tBuzWarn5RestTm ACCESS p_NtParamBuzWarn5RestTm;
	p_usiBuzWarn5OnCntr ACCESS p_NtParamBuzWarn5OnCntr;
	p_bBuzWarn5StopSeqEn ACCESS p_NtParamBuzWarn5StopSeqEn;
	p_usiBuzWarn5StopSeqCntr ACCESS p_NtParamBuzWarn5StopSeqCntr;

	p_tBuzAlertOnTm ACCESS p_NtParamBuzAlertOnTm;
	p_tBuzAlertRestTm ACCESS p_NtParamBuzAlertRestTm;
	p_usiBuzAlertOnCntr ACCESS p_NtParamBuzAlertOnCntr;
	p_bBuzAlertStopSeqEn ACCESS p_NtParamBuzAlertStopSeqEn;
	p_usiBuzAlertStopSeqCntr ACCESS p_NtParamBuzAlertStopSeqCntr;

	p_tTLBlueBlinkTm ACCESS p_NtParamTLBlueBlinkTm;
	p_tTLAmberBlinkTm ACCESS p_NtParamTLAmberBlinkTm;
	p_tTLWhiteBlinkTm ACCESS p_NtParamTLWhiteBlinkTm;
	p_tTLRedBlinkTm ACCESS p_NtParamTLRedBlinkTm;
	p_tTLGreenBlinkTm ACCESS p_NtParamTLGreenBlinkTm;

	//  ----------------------------------------------  ||  ---------------------------------------------	//

	p_bCoverSwitchSig ACCESS p_DICoverSWSig;
	p_eTLBuzMode ACCESS p_NtParamTLBuzMode;

	p_bMcParamAGVComEn ACCESS p_McParamAGVComEn; //Add

	p_tyBuffer1BffrStat ACCESS p_Buffer1BffrStat; //ADD
	p_tyBuffer2BffrStat ACCESS p_Buffer2BffrStat; //ADD
	p_tyBuffer3BffrStat ACCESS p_Buffer3BffrStat; //ADD
	(* Always Change If Project Change *)
	p_eMcParamMagExMode ACCESS p_McParamMagExMode;
END_ACTION
```

#### Act_Link.st
```iecst
(** 2019-03-29 **)
ACTION Act_Link:

	p_bWarning			:= p_bLinkAlarmWarning OR (p_bLinkAlarmInfo AND NOT (p_bLinkAlarmInfoLF AND p_bLinkLFBuzMute) AND
													NOT(p_bLinkMagFullInfo AND p_bLinkMagFullTLMuteBuzz));

	p_bWarningNoBuz		:= (p_bLinkAlarmInfoLF AND p_bLinkLFBuzMute) OR (p_bLinkAlarmInfo AND p_bLinkMagFullInfo AND p_bLinkMagFullTLMuteBuzz);

END_ACTION
```

### Alarm.var
```iecst
(*2019-03-25*)
(**)
(*Constant*)
VAR CONSTANT
	c_udiAlarmCurrMax : UDINT := 200;
	c_udiAlarmHistoryMax : UDINT := 300;
END_VAR
(**)
(*Action & State & Status*)
VAR
	p_AlarmStat : UDINT;
	p_AlarmStatus : UDINT;
	p_AlarmStatTxt : UDINT;
END_VAR
(**)
(*Alarm*)
(**)
(*Output*)
VAR
	p_AlarmErr : UDINT;
	p_AlarmWarning : UDINT;
	p_AlarmCurrList : UDINT;
	p_AlarmRecoveryList : UDINT;
	p_AlarmHistoryList : UDINT;
	p_AlarmInfo : UDINT;
	p_AlarmInfoLF : UDINT;
	p_AlarmInfoMsg : UDINT;
	p_AlarmHistoryFileNotFound : UDINT;
END_VAR
(**)
(*Alarm Program Name: Declare Global Variables Based on the Projects' Packages.*)
VAR
	g_sAWOpenProgNm : STRING[15];
	g_sAWCloseProgNm : STRING[15];
	g_sMagAWOpenProgNm : STRING[15];
	g_sTravProgNm : STRING[15];
	g_sLifterBtmProgNm : STRING[15];
	g_sConvProgNm : STRING[15];
	g_sDCConvProgNm : STRING[15];
	g_sMagConvProgNm : STRING[15];
	g_sMagConv2ClpProgNm : STRING[15];
	g_sBufferProgNm : STRING[15];
	g_sMotorBrkProgNm : STRING[15];
	g_sMtrPshrProgNm : STRING[15];
	g_sStepperProgNm : STRING[15];
	g_sPneuNoSenProgNm : STRING[15];
	g_sPneuExtSenProgNm : STRING[15];
	g_sPneuRetSenProgNm : STRING[15];
	g_sPneu2SenProgNm : STRING[15];
	g_sPneu3SenProgNm : STRING[15];
	g_sUSSMEMAProgNm : STRING[15];
	g_sDSSMEMAProgNm : STRING[15];
	g_sHermesProgNm : STRING[15];
	g_sUSHermesProgNm : STRING[15];
	g_sDSHermesAProgNm : STRING[15];
	g_sDSHermesBProgNm : STRING[15];
	g_sRmtHermesProgNm : STRING[15];
	g_sSvyHermesProgNm : STRING[15];
	g_sLFLeaderProgNm : STRING[15];
	g_sLFFollowerProgNm : STRING[15];
	g_sLCSProgNm : STRING[15];
	g_sLCSLFProgNm : STRING[15];
	g_sLCSMngRcpProgNm : STRING[15];
	g_sTCPProgNm : STRING[15];
	g_sUSSOTProgNm : STRING[15];
	g_sDSSOTProgNm : STRING[15];
	g_sBarcodeRdrProgNm : STRING[15];
	g_sRS232MirtecProgNm : STRING[15];
	g_sProdRcpProgNm : STRING[15];
	g_sMagRcpProgNm : STRING[15];
	g_sMpProdRcpProgNm : STRING[15];
	g_sAlarmProgNm : STRING[15];
	g_sNtParamProgNm : STRING[15];
	g_sMcParamProgNm : STRING[15];
	g_sUsrMgmtProgNm : STRING[15];
	g_sLibVerProgNm : STRING[15];
	g_sUsrFolderProgNm : STRING[15];
	g_sHWInfoProgNm : STRING[15];
	g_sDInputProgNm : STRING[15];
	g_sTimeProgNm : STRING[15];
	g_sMachineProgNm : STRING[15];
	g_sOps1ProgNm : STRING[15];
	g_sOpsTravLifULProgNm : STRING[15];
	g_sOpsMagConvULProgNm : STRING[15];
	g_sOpsMagConvUL2ProgNm : STRING[15];
	g_sOpsMagConvUL3ProgNm : STRING[15];
	g_sOpsLifMagULProgNm : STRING[15];
	g_sOpsInMagConvProgNm : STRING[15];
	g_sOpsOutMagConvProgNm : STRING[15];
	g_sOpsMagConvStprProgNm : STRING[15];
	g_sOpsMagConvStpr2ProgNm : STRING[15];
	g_sWarningLibVersion : STRING[15];
	g_sAGVComProgNm : STRING[15];
	g_sAGVProgNm : STRING[15];
	g_sLiberWarnName : STRING[15];
	g_sSimu1ProgNm : STRING[15];
	g_sFrameProgNm : STRING[15];
	g_sOpsTravLifLDProgNm : STRING[15];
	g_sOpsMagConvLDProgNm : STRING[15];
	g_sOpsLifMagLDProgNm : STRING[15];
	g_sAutoRcpProgNm : STRING[15];
END_VAR
```

### Program Logical/Alarm/Alarm

#### InputRef_Link.var
```iecst
(*2019-01-07*)
(**)
(*External Data*)
VAR
	p_tyLinkUsrFolderAlmData : REFERENCE TO tyAlmDat;
	p_tyLinkLibVerAlmData : REFERENCE TO tyAlmDat;
	p_tyLinkTimeAlmData : REFERENCE TO tyAlmDat;
	p_tyLinkTimeAlmData1 : REFERENCE TO tyAlmDat;
	p_tyLinkHWInfoAlmData : REFERENCE TO tyAlmDat;
	p_tyLinkProdRcpAlmData : REFERENCE TO tyAlmDat;
	p_tyLinkMpProdRcpAlmData : REFERENCE TO tyAlmDat;
	p_tyLinkMagRcpAlmData : REFERENCE TO tyAlmDat;
	p_tyLinkMagRcpAlmData1 : REFERENCE TO tyAlmDat;
	p_tyLinkMcParamAlmData : REFERENCE TO tyAlmDat;
	p_tyLinkNtParamAlmData : REFERENCE TO tyAlmDat;
	p_tyLinkUsrMgmtAlmData : REFERENCE TO tyAlmDat;
	p_tyLinkBuffer1AlmData : REFERENCE TO tyAlmDat;
	p_tyLinkBuffer2AlmData : REFERENCE TO tyAlmDat;
	p_tyLinkBuffer3AlmData : REFERENCE TO tyAlmDat;
	p_tyLinkBuffer4AlmData : REFERENCE TO tyAlmDat;
	p_tyLinkUSSMEMA1AlmData : REFERENCE TO tyAlmDat;
	p_tyLinkUSSMEMA2AlmData : REFERENCE TO tyAlmDat;
	p_tyLinkUSSMEMA3AlmData : REFERENCE TO tyAlmDat;
	p_tyLinkUSSMEMA4AlmData : REFERENCE TO tyAlmDat;
	p_tyLinkDSSMEMA1AlmData : REFERENCE TO tyAlmDat;
	p_tyLinkDSSMEMA2AlmData : REFERENCE TO tyAlmDat;
	p_tyLinkDSSMEMA3AlmData : REFERENCE TO tyAlmDat;
	p_tyLinkDSSMEMA4AlmData : REFERENCE TO tyAlmDat;
	p_tyLinkDSSMEMAAAlmData : REFERENCE TO tyAlmDat;
	p_tyLinkDSSMEMABAlmData : REFERENCE TO tyAlmDat;
	p_tyLinkInShutterAlmData : REFERENCE TO tyAlmDat;
	p_tyLinkOutShutterAlmData : REFERENCE TO tyAlmDat;
	p_tyLinkPullerAlmData : REFERENCE TO tyAlmDat;
	p_tyLinkPullConvAlmData : REFERENCE TO tyAlmDat;
	p_tyLinkMagConv1AlmData : REFERENCE TO tyAlmDat;
	p_tyLinkMagConv2AlmData : REFERENCE TO tyAlmDat;
	p_tyLinkMagConv3AlmData : REFERENCE TO tyAlmDat;
	p_tyLinkMagConv4AlmData : REFERENCE TO tyAlmDat;
	p_tyLinkAWOpenAlmData : REFERENCE TO tyAlmDat;
	p_tyLinkAWOpenAlmData1 : REFERENCE TO tyAlmDat;
	p_tyLinkAWOpenAlmData2 : REFERENCE TO tyAlmDat;
	p_tyLinkAWOpenAlmData3 : REFERENCE TO tyAlmDat;
	p_tyLinkTravAlmData : REFERENCE TO tyAlmDat;
	p_tyLinkTravAlmData1 : REFERENCE TO tyAlmDat;
	p_tyLinkTravAlmData2 : REFERENCE TO tyAlmDat;
	p_tyLinkTravAlmData3 : REFERENCE TO tyAlmDat;
	p_tyLinkLifterBtmAlmData : REFERENCE TO tyAlmDat;
	p_tyLinkLifterBtmAlmData1 : REFERENCE TO tyAlmDat;
	p_tyLinkLifterBtmAlmData2 : REFERENCE TO tyAlmDat;
	p_tyLinkLifterBtmAlmData3 : REFERENCE TO tyAlmDat;
	p_tyLinkDIAlmData1 : REFERENCE TO tyAlmDat;
	p_tyLinkDIAlmData2 : REFERENCE TO tyAlmDat;
	p_tyLinkDIAlmData3 : REFERENCE TO tyAlmDat;
	p_tyLinkDIAlmData4 : REFERENCE TO tyAlmDat;
	p_tyLinkDIAlmData5 : REFERENCE TO tyAlmDat;
	p_tyLinkDIAlmData6 : REFERENCE TO tyAlmDat;
	p_tyLinkAGVAlmData1 : REFERENCE TO tyAlmDat;
	p_tyLinkAGVMag1AlmData : REFERENCE TO tyAlmDat;
	p_tyLinkAGVMag2AlmData : REFERENCE TO tyAlmDat;
	p_tyLinkAGVMag3AlmData : REFERENCE TO tyAlmDat;
	p_tyLinkAGVMag4AlmData : REFERENCE TO tyAlmDat;
	p_tyLinkHermesAlmData : REFERENCE TO tyAlmDat;
	p_tyLinkDSHermesAAlmData : REFERENCE TO tyAlmDat;
	p_tyLinkDSHermesAAlmData1 : REFERENCE TO tyAlmDat;
	p_tyLinkDSHermesAAlmData2 : REFERENCE TO tyAlmDat;
	p_tyLinkDSHermesAAlmData3 : REFERENCE TO tyAlmDat;
	p_tyLinkDSHermesAAlmData4 : REFERENCE TO tyAlmDat;
	p_tyLinkDSHermesBAlmData : REFERENCE TO tyAlmDat;
	p_tyLinkDSHermesBAlmData1 : REFERENCE TO tyAlmDat;
	p_tyLinkDSHermesBAlmData2 : REFERENCE TO tyAlmDat;
	p_tyLinkDSHermesBAlmData3 : REFERENCE TO tyAlmDat;
	p_tyLinkDSHermesBAlmData4 : REFERENCE TO tyAlmDat;
	p_tyLinkRmtHermesAlmData : REFERENCE TO tyAlmDat;
	p_tyLinkRmtHermesAlmData1 : REFERENCE TO tyAlmDat;
	p_tyLinkRmtHermesAlmData2 : REFERENCE TO tyAlmDat;
	p_tyLinkRmtHermesAlmData3 : REFERENCE TO tyAlmDat;
	p_tyLinkLFLeaderAlmData : REFERENCE TO tyAlmDat;
	p_tyLinkLFFollowerAlmData : REFERENCE TO tyAlmDat;
	p_tyLinkLFFollowerInfoData : REFERENCE TO tyAlmDat;
	p_tyLinkLFFollowerInfoData1 : REFERENCE TO tyAlmDat;
	p_tyLinkFollower1AlmData : REFERENCE TO tyAlmDat;
	p_tyLinkFollower1InfoData : REFERENCE TO tyAlmDat;
	p_tyLinkFollower1InfoData1 : REFERENCE TO tyAlmDat;
	p_tyLinkFollower2AlmData : REFERENCE TO tyAlmDat;
	p_tyLinkFollower2InfoData : REFERENCE TO tyAlmDat;
	p_tyLinkFollower2InfoData1 : REFERENCE TO tyAlmDat;
	p_tyLinkLCSMngRcpAlmData : REFERENCE TO tyAlmDat;
	p_tyLinkLCSLFAlmData : REFERENCE TO tyAlmDat;
	p_tyLinkLCSLFInfoData : REFERENCE TO tyAlmDat;
	p_tyLinkOpsTravLifLDAlmData : REFERENCE TO tyAlmDat;
	p_tyLinkOpsMagLD1AlmData : REFERENCE TO tyAlmDat;
	p_tyLinkOpsMagLD1AlmData1 : REFERENCE TO tyAlmDat;
	p_tyLinkOpsMagLD2AlmData : REFERENCE TO tyAlmDat;
	p_tyLinkOpsMagLD2AlmData1 : REFERENCE TO tyAlmDat;
	p_tyLinkOpsMagLD3AlmData : REFERENCE TO tyAlmDat;
	p_tyLinkOpsMagLD3AlmData1 : REFERENCE TO tyAlmDat;
	p_tyLinkOpsMagLD4AlmData : REFERENCE TO tyAlmDat;
	p_tyLinkOpsMagLD4AlmData1 : REFERENCE TO tyAlmDat;
	p_tyLinkOpsMagConvLD1AlmData : REFERENCE TO tyAlmDat;
	p_tyLinkOpsMagConvLD1AlmData1 : REFERENCE TO tyAlmDat;
	p_tyLinkOpsMagConvLD2AlmData : REFERENCE TO tyAlmDat;
	p_tyLinkOpsMagConvLD2AlmData1 : REFERENCE TO tyAlmDat;
	p_tyLinkOpsMagConvLD3AlmData : REFERENCE TO tyAlmDat;
	p_tyLinkOpsMagConvLD3AlmData1 : REFERENCE TO tyAlmDat;
	p_tyLinkOpsMagConvLD4AlmData : REFERENCE TO tyAlmDat;
	p_tyLinkOpsMagConvLD4AlmData1 : REFERENCE TO tyAlmDat;
	p_tyLinkSelClamp1AlmData : REFERENCE TO tyAlmDat;
	p_tyLinkSelClamp2AlmData : REFERENCE TO tyAlmDat;
	p_tyLinkSelClamp3AlmData : REFERENCE TO tyAlmDat;
	p_tyLinkSelClamp4AlmData : REFERENCE TO tyAlmDat;
	p_tyLinkUSSOT1AlmData : REFERENCE TO tyAlmDat;
	p_tyLinkUSSOT2AlmData : REFERENCE TO tyAlmDat;
	p_tyLinkUSSOT3AlmData : REFERENCE TO tyAlmDat;
	p_tyLinkUSSOT4AlmData : REFERENCE TO tyAlmDat;
	p_tyLinkDSSOT1AlmData : REFERENCE TO tyAlmDat;
	p_tyLinkDSSOT2AlmData : REFERENCE TO tyAlmDat;
	p_tyLinkDSSOT3AlmData : REFERENCE TO tyAlmDat;
	p_tyLinkDSSOT4AlmData : REFERENCE TO tyAlmDat;
	p_tyLinkMcAlarmData : REFERENCE TO tyAlmDat;
	p_tyLinkMc1AlarmData : REFERENCE TO tyAlmDat;
	p_tyLinkUSBBarcodeAlmData : REFERENCE TO tyAlmDat;
	p_tyLinkUSBBarcodeAlmData1 : REFERENCE TO tyAlmDat;
	p_tyLinkUSBBarcodeAlmData2 : REFERENCE TO tyAlmDat;
	p_tyLinkRS232FrmAlmData : REFERENCE TO tyAlmDat;
	p_tyLinkAWPushOrPullerAlmData : REFERENCE TO tyAlmDat;
	p_tyLinkAWPushOrPullerAlmData1 : REFERENCE TO tyAlmDat;
	p_tyLinkAWPushOrPullerAlmData2 : REFERENCE TO tyAlmDat;
	p_tyLinkAWPushOrPullerAlmData3 : REFERENCE TO tyAlmDat;
	p_tyLinkMtrPshrAlmData : REFERENCE TO tyAlmDat;
	p_tyLinkOpsLifMagLDAlmData : REFERENCE TO tyAlmDat;
	p_tyLinkOpsLifMagLDAlmData1 : REFERENCE TO tyAlmDat;
	p_tyLinkPPAlmData : REFERENCE TO tyAlmDat;
	p_tyLinkPPAlmData1 : REFERENCE TO tyAlmDat;
	p_tyLinkPPAlmData2 : REFERENCE TO tyAlmDat;
	p_tyLinkPPAlmData3 : REFERENCE TO tyAlmDat;
	p_tyLinkInShutterAlmData2 : REFERENCE TO tyAlmDat;
	p_tyLinkInShutterAlmData3 : REFERENCE TO tyAlmDat;
	p_tyLinkUSHermesInfoData1 : REFERENCE TO tyAlmDat;
	p_tyLinkUSHermesInfoData2 : REFERENCE TO tyAlmDat;
	p_tyLinkRmtHermesInfoData : REFERENCE TO tyAlmDat;
	p_tyLinkSvyHermesAlmData : REFERENCE TO tyAlmDat;
	p_tyLinkSvyHermesAlmData1 : REFERENCE TO tyAlmDat;
	p_tyLinkSvyHermesAlmData2 : REFERENCE TO tyAlmDat;
	p_tyLinkSvyHermesAlmData3 : REFERENCE TO tyAlmDat;
	p_tyLinkSvyHermesAlmData4 : REFERENCE TO tyAlmDat;
	p_tyLinkSvyHermesInfoData : REFERENCE TO tyAlmDat;
	p_tyLinkSvyHermesInfoData1 : REFERENCE TO tyAlmDat;
	p_tyLinkSvyHermesInfoData2 : REFERENCE TO tyAlmDat;
	p_tyLinkSvyHermesInfoData3 : REFERENCE TO tyAlmDat;
	p_tyLinkSvyHermesInfoData4 : REFERENCE TO tyAlmDat;
	p_tyLinkOutShutterAlmData2 : REFERENCE TO tyAlmDat;
	p_tyLinkTrllyAlmData : REFERENCE TO tyAlmDat;
	p_tyLinkTrlly2AlmData : REFERENCE TO tyAlmDat;
	p_tyLinkAutoRcpAlmData : REFERENCE TO tyAlmDat;
	p_tyLinkAutoRcpInfoData : REFERENCE TO tyAlmDat;
	p_tyLinkAutoRcpInfoData1 : REFERENCE TO tyAlmDat;
END_VAR
```

#### Local.var
```iecst
(*2019-05-09*)
(**)
(*Local Action, State & Status*)
VAR
	eAct : eAlarmAction := AlarmActIdle;
	eStat : eAlarmAction := AlarmActIdle;
	eStatus : eFBStatus := Idle;
	udiStatus : UDINT := 0;
	sStatTxt : STRING[200] := '';
	a_sStatText : ARRAY[0..50] OF STRING[200] := ['Idling','Creating Directory','Deleting Old Alarm Log File','Reading History File','Writing History File','Appending Alarm Log File','Appending Alarm Log File & Writing History File','Resetting History','Background Start Alarm Log','Background Stop Alarm Log',41('')];
END_VAR
(**)
(*Local Alarm*)
VAR
	tyAlmData : tyAlmDat;
	a_tyAlmText : ARRAY[10000..10099] OF tyAlmTxt := [(sAlmText:='Create User Directory Error',sRcyText:='An Error Occurred While Attempting To Create User Directory. Please Contact Nutek For A Possible Solution'),(sAlmText:='Create Alarm Directory Error',sRcyText:='An Error Occurred While Attempting To Create Alarm Directory. Please Contact Nutek For A Possible Solution'),(sAlmText:='Get Directory Info Error While Deleting Old Log',sRcyText:='An Error Was Encountered While Getting Directory Info. Please Contact Nutek For A Possible Solution.'),(sAlmText:='Directory Read Error While Deleting Old Log',sRcyText:='An Error Was Encountered While Reading Directory. Please Contact Nutek For A Possible Solution.'),(sAlmText:='File Delete Error While Deleting Old Log',sRcyText:='An Error Was Encountered While Trying To Delete File. Please Contact Nutek For A Possible Solution.'),(sAlmText:='File Open Error While Reading Alarm History',sRcyText:='An Error Was Encountered While Trying To Open File. Please Contact Nutek For A Possible Solution.'),(sAlmText:='File Read Error While Reading Alarm History',sRcyText:='An Error Was Encountered While Trying To Read File. Please Contact Nutek For A Possible Solution.'),(sAlmText:='File Close Error While Reading Alarm History',sRcyText:='An Error Was Encountered While Trying To Close File. Please Contact Nutek For A Possible Solution.'),(sAlmText:='File Open Error While Writing Alarm History',sRcyText:='An Error Was Encountered While Trying To Open File. Please Contact Nutek For A Possible Solution.'),(sAlmText:='File Create Error While Writing Alarm History',sRcyText:='An Error Was Encountered While Trying To Create File. Please Contact Nutek For A Possible Solution.'),(sAlmText:='File Write Error While Writing Alarm History',sRcyText:='An Error Was Encountered While Trying To Write File. Please Contact Nutek For A Possible Solution.'),(sAlmText:='File Close Error While Writing Alarm History',sRcyText:='An Error Was Encountered While Trying To Close File. Please Contact Nutek For A Possible Solution.'),(sAlmText:='Directory Does Not Exist While Writing Alarm History',sRcyText:='The Directory Does Not Exist. Please Contact Nutek For A Possible Solution.'),(sAlmText:='File Open Error While Writing Alarm Log',sRcyText:='An Error Was Encountered While Trying To Open File. Please Contact Nutek For A Possible Solution.'),(sAlmText:='File Create Error While Writing Alarm Log',sRcyText:='An Error Was Encountered While Trying To Create File. Please Contact Nutek For A Possible Solution.'),(sAlmText:='Get File Info Error While Writing Alarm Log',sRcyText:='An Error Was Encountered While Getting File Info. Please Contact Nutek For A Possible Solution.'),(sAlmText:='File Write Error While Writing Alarm Log',sRcyText:='An Error Was Encountered While Trying To Write File. Please Contact Nutek For A Possible Solution.'),(sAlmText:='File Close Error While Writing Alarm Log',sRcyText:='An Error Was Encountered While Trying To Close File. Please Contact Nutek For A Possible Solution.'),(sAlmText:='Directory Does Not Exist While Writing Alarm Log',sRcyText:='The Directory Does Not Exist. Please Contact Nutek For A Possible Solution.'),(sAlmText:='File Open Error While Writing Alarm History',sRcyText:='An Error Was Encountered While Trying To Open File. Please Contact Nutek For A Possible Solution.'),(sAlmText:='File Create Error While Writing Alarm History',sRcyText:='An Error Was Encountered While Trying To Create File. Please Contact Nutek For A Possible Solution.'),(sAlmText:='File Write Error While Writing Alarm History',sRcyText:='An Error Was Encountered While Trying To Write File. Please Contact Nutek For A Possible Solution.'),(sAlmText:='File Close Error While Writing Alarm History',sRcyText:='An Error Was Encountered While Trying To Close File. Please Contact Nutek For A Possible Solution.'),(sAlmText:='Directory Does Not Exist While Writing Alarm History',sRcyText:='The Directory Does Not Exist. Please Contact Nutek For A Possible Solution.'),(sAlmText:='File Open Error While Writing Alarm Log',sRcyText:='An Error Was Encountered While Trying To Open File. Please Contact Nutek For A Possible Solution.'),(sAlmText:='File Create Error While Writing Alarm Log',sRcyText:='An Error Was Encountered While Trying To Create File. Please Contact Nutek For A Possible Solution.'),(sAlmText:='Get File Info Error While Writing Alarm Log',sRcyText:='An Error Was Encountered While Getting File Info. Please Contact Nutek For A Possible Solution.'),(sAlmText:='File Write Error While Writing Alarm Log',sRcyText:='An Error Was Encountered While Trying To Write File. Please Contact Nutek For A Possible Solution.'),(sAlmText:='File Close Error While Writing Alarm Log',sRcyText:='An Error Was Encountered While Trying To Close File. Please Contact Nutek For A Possible Solution.'),(sAlmText:='Directory Does Not Exist While Writing Alarm Log',sRcyText:='The Directory Does Not Exist. Please Contact Nutek For A Possible Solution.'),(sAlmText:='File Open Error While Resetting Alarm History',sRcyText:='An Error Was Encountered While Trying To Open File. Please Contact Nutek For A Possible Solution.'),(sAlmText:='File Create Error While Resetting Alarm History',sRcyText:='An Error Was Encountered While Trying To Create File. Please Contact Nutek For A Possible Solution.'),(sAlmText:='File Write Error While Resetting Alarm History',sRcyText:='An Error Was Encountered While Trying To Write File. Please Contact Nutek For A Possible Solution.'),(sAlmText:='File Close Error While Resetting Alarm History',sRcyText:='An Error Was Encountered While Trying To Close File. Please Contact Nutek For A Possible Solution.'),(sAlmText:='Directory Does Not Exist While Resetting Alarm History',sRcyText:='The Directory Does Not Exist. Please Contact Nutek For A Possible Solution.'),65((0))];
END_VAR
(**)
(*Local Output*)
VAR
	bErr : BOOL;
	bWarning : BOOL;
	a_tyCurrList : ARRAY[1..c_udiAlarmCurrMax] OF tyAlarmCurr;
	a_sRecoveryList : ARRAY[1..c_udiAlarmCurrMax] OF STRING[200];
	a_udiRecoveryList : ARRAY[1..c_udiAlarmCurrMax] OF UDINT;
	a_sHistoryList : ARRAY[1..c_udiAlarmHistoryMax] OF STRING[200];
	bInfo : BOOL;
	sInfoMsg : STRING[200];
	bHistoryFileNotFound : BOOL;
	bInfoLF : BOOL := FALSE;
END_VAR
(**)
(*Local Input*)
VAR
	udiRstErr : UDINT := 0;
	dtCurrDT : DATE_AND_TIME;
	a_tyAlmData : ARRAY[1..c_udiAlarmCurrMax] OF tyAlmDat;
	udiFileKeepDay : UDINT := 30;
	sProgNm : STRING[15] := 'Alarm';
	bNtSettingsLoadDone : BOOL := TRUE;
END_VAR
(**)
(*Local*)
VAR
	bRstErr : BOOL;
	udiRstErrOld : UDINT;
	bInitDone : BOOL;
	bInitialDone : BOOL;
	bAlarmLog : BOOL;
	usiStep : USINT;
	udi : UDINT;
	iInfoCntr : INT;
	sAlmMsg : STRING[300];
	udiAlmCntr : UDINT;
	udiAlmRecvryCntr : UDINT;
	udiLogCntr : UDINT;
	udiWriteLogCntr : UDINT;
	a_sLogList : ARRAY[1..c_udiAlarmCurrMax] OF STRING[200];
	bAlmUpdt : BOOL;
	dtCurrDTTemp : DATE_AND_TIME;
	a_udiRunTimeOld : ARRAY[1..c_udiAlarmCurrMax] OF UDINT;
	fbDirCreate1 : fbDirCreate;
	fbDirCreate2 : fbDirCreate;
	fbFileAppend1 : fbFileFullAppend;
	fbFileOldDel1 : fbFileOldDel;
	fbFileRead1 : fbFileFullRead;
	fbFileWrite1 : fbFileFullWrite;
	udi1 : UDINT;
	udi2 : UDINT;
	udiRecorded : ARRAY[1..c_udiAlarmCurrMax] OF UDINT;
	udiRecorded1 : UDINT;
	bRstWarning : BOOL;
	udiWarningMax : UDINT := 1;
	sWarningMsg : STRING[300];
	sWarningID : STRING[80] := '';
	sWarningCompareMsg : STRING[300];
	a_tyWarningCurrList : ARRAY[1..c_udiAlarmCurrMax] OF tyAlarmCurr;
	a_tyHistoryList : ARRAY[1..c_udiAlarmHistoryMax] OF tyHistory;
	WarningListOccur : BOOL := TRUE;
	udiErrorCode : UDINT;
	fbDeleteLogTmr : TON := (PT:=T#24h);
	fbDlyTmr : TON := (PT:=T#5s);
	sDT : STRING[80];
	udiModuleNum : UDINT := 5051;
END_VAR
```

#### Act_InitGlobal.st
```iecst
(** 2019-03-25 **)
ACTION Act_InitGlobal:

	(* Always Change If Project Change *)

	//Pass Data To Link
	p_tyLinkUsrFolderAlmData ACCESS p_UsrFolderAlmData;
	p_tyLinkLibVerAlmData ACCESS p_LibVerAlmData;
	p_tyLinkTimeAlmData ACCESS p_TimeAlmData;
	p_tyLinkTimeAlmData1 ACCESS p_TimeAlmData1;
	p_tyLinkHWInfoAlmData ACCESS p_HWInfoAlmData;
	p_tyLinkProdRcpAlmData ACCESS p_ProdRcpAlmData;
	p_tyLinkMpProdRcpAlmData ACCESS p_MpProdRcpAlmData;
	p_tyLinkMagRcpAlmData ACCESS p_MagRcpAlmData;
	p_tyLinkMagRcpAlmData1 ACCESS p_MagRcpAlmData1;
	p_tyLinkMcParamAlmData ACCESS p_McParamAlmData;
	p_tyLinkNtParamAlmData ACCESS p_NtParamAlmData;
	p_tyLinkUsrMgmtAlmData ACCESS p_UsrMgmtAlmData;
	p_tyLinkBuffer1AlmData ACCESS p_Buffer1AlmData;
	p_tyLinkBuffer2AlmData ACCESS p_Buffer2AlmData;
	p_tyLinkBuffer3AlmData ACCESS p_Buffer3AlmData;
	p_tyLinkBuffer4AlmData ACCESS p_Buffer4AlmData;
	p_tyLinkUSSMEMA1AlmData ACCESS p_USSMEMA1AlmData;
	p_tyLinkUSSMEMA2AlmData ACCESS p_USSMEMA2AlmData;
	p_tyLinkUSSMEMA3AlmData ACCESS p_USSMEMA3AlmData;
	p_tyLinkUSSMEMA4AlmData ACCESS p_USSMEMA4AlmData;
	p_tyLinkDSSMEMA1AlmData ACCESS p_DSSMEMA1AlmData;
	p_tyLinkDSSMEMA2AlmData ACCESS p_DSSMEMA2AlmData;
	p_tyLinkDSSMEMA3AlmData ACCESS p_DSSMEMA3AlmData;
	p_tyLinkDSSMEMA4AlmData ACCESS p_DSSMEMA4AlmData;
	p_tyLinkDSSMEMAAAlmData ACCESS p_DSSMEMAAAlmData;
	p_tyLinkDSSMEMABAlmData ACCESS p_DSSMEMABAlmData;
	p_tyLinkInShutterAlmData ACCESS p_Pneu2SenInShutterAlmData;
	p_tyLinkOutShutterAlmData ACCESS p_Pneu2SenOutShutterAlmData;
	p_tyLinkPullerAlmData ACCESS p_Pneu2SenPullerAlmData;
	p_tyLinkPullConvAlmData ACCESS p_PullConvAlmData;
	p_tyLinkMagConv1AlmData ACCESS p_MagConv2Clp1AlmData;
	p_tyLinkMagConv2AlmData ACCESS p_MagConv2Clp2AlmData;
	p_tyLinkMagConv3AlmData ACCESS p_MagConv2Clp3AlmData;
	p_tyLinkMagConv4AlmData ACCESS p_MagConv2Clp4AlmData;
	p_tyLinkAWOpenAlmData ACCESS p_AWOpenAlmData;
	p_tyLinkAWOpenAlmData1 ACCESS p_AWOpenAlmData1;
	p_tyLinkAWOpenAlmData2 ACCESS p_AWOpenAlmData2;
	p_tyLinkAWOpenAlmData3 ACCESS p_AWOpenAlmData3;
	p_tyLinkTravAlmData ACCESS p_TravAlmData;
	p_tyLinkTravAlmData1 ACCESS p_TravAlmData1;
	p_tyLinkTravAlmData2 ACCESS p_TravAlmData2;
	p_tyLinkTravAlmData3 ACCESS p_TravAlmData3;
	p_tyLinkLifterBtmAlmData ACCESS p_LifterBtmAlmData;
	p_tyLinkLifterBtmAlmData1 ACCESS p_LifterBtmAlmData1;
	p_tyLinkLifterBtmAlmData2 ACCESS p_LifterBtmAlmData2;
	p_tyLinkLifterBtmAlmData3 ACCESS p_LifterBtmAlmData3;
	p_tyLinkDIAlmData1 ACCESS p_DIAlmData1;
	p_tyLinkDIAlmData2 ACCESS p_DIAlmData2;
	p_tyLinkDIAlmData3 ACCESS p_DIAlmData3;
	p_tyLinkDIAlmData4 ACCESS p_DIAlmData4;
	p_tyLinkDIAlmData5 ACCESS p_DIAlmData5;
	p_tyLinkDIAlmData6 ACCESS p_DIAlmData6;		//JOHN
	p_tyLinkAGVMag1AlmData ACCESS p_AGVMag1AlmData;
	p_tyLinkAGVMag2AlmData ACCESS p_AGVMag2AlmData;
	p_tyLinkAGVMag3AlmData ACCESS p_AGVMag3AlmData;
	p_tyLinkAGVMag4AlmData ACCESS p_AGVMag4AlmData;
	p_tyLinkHermesAlmData ACCESS p_HermesAlmData;
	p_tyLinkDSHermesAAlmData ACCESS p_DSHermesAAlmData;
	p_tyLinkDSHermesAAlmData1 ACCESS p_DSHermesAAlmData1;
	p_tyLinkDSHermesAAlmData2 ACCESS p_DSHermesAAlmData2;
	p_tyLinkDSHermesAAlmData3 ACCESS p_DSHermesAAlmData3;
	p_tyLinkDSHermesAAlmData4 ACCESS p_DSHermesAAlmData4;
	p_tyLinkDSHermesBAlmData ACCESS p_DSHermesBAlmData;
	p_tyLinkDSHermesBAlmData1 ACCESS p_DSHermesBAlmData1;
	p_tyLinkDSHermesBAlmData2 ACCESS p_DSHermesBAlmData2;
	p_tyLinkDSHermesBAlmData3 ACCESS p_DSHermesBAlmData3;
	p_tyLinkDSHermesBAlmData4 ACCESS p_DSHermesBAlmData4;
	p_tyLinkRmtHermesAlmData ACCESS p_RmtHermesAlmData;
	p_tyLinkRmtHermesAlmData1 ACCESS p_RmtHermesAlmData1;
	p_tyLinkRmtHermesAlmData2 ACCESS p_RmtHermesAlmData2;
	p_tyLinkRmtHermesAlmData3 ACCESS p_RmtHermesAlmData3;
	p_tyLinkLFLeaderAlmData ACCESS p_LFLeaderAlmData;
	p_tyLinkLFFollowerAlmData ACCESS p_LFFollowerAlmData;
	p_tyLinkLFFollowerInfoData ACCESS p_LFFollowerInfoData;
	p_tyLinkLFFollowerInfoData1 ACCESS p_LFFollowerInfoData1;
	p_tyLinkFollower1AlmData ACCESS p_Follower1AlmData;
	p_tyLinkFollower1InfoData ACCESS p_Follower1InfoData;
	p_tyLinkFollower1InfoData1 ACCESS p_Follower1InfoData1;
	p_tyLinkFollower2AlmData ACCESS p_Follower2AlmData;
	p_tyLinkFollower2InfoData ACCESS p_Follower2InfoData;
	p_tyLinkFollower2InfoData1 ACCESS p_Follower2InfoData1;
	p_tyLinkLCSMngRcpAlmData ACCESS p_LCSMngRcpAlmData;
	p_tyLinkLCSLFAlmData ACCESS p_LCSLFAlmData;
	p_tyLinkLCSLFInfoData ACCESS p_LCSLFInfoData;
	p_tyLinkOpsTravLifLDAlmData ACCESS p_OpsTravLifLDAlmData;
//	p_tyLinkOpsMagLD1AlmData ACCESS p_OpsMagLD1AlmData;
//	p_tyLinkOpsMagLD1AlmData1 ACCESS p_OpsMagLD1AlmData1;
//	p_tyLinkOpsMagLD2AlmData ACCESS p_OpsMagLD2AlmData;
//	p_tyLinkOpsMagLD2AlmData1 ACCESS p_OpsMagLD2AlmData1;
//	p_tyLinkOpsMagLD3AlmData ACCESS p_OpsMagLD3AlmData;
//	p_tyLinkOpsMagLD3AlmData1 ACCESS p_OpsMagLD3AlmData1;
//	p_tyLinkOpsMagLD4AlmData ACCESS p_OpsMagLD4AlmData;
//	p_tyLinkOpsMagLD4AlmData1 ACCESS p_OpsMagLD4AlmData1;
	p_tyLinkOpsMagConvLD1AlmData ACCESS p_OpsMagConvLD1AlmData;
	p_tyLinkOpsMagConvLD1AlmData1 ACCESS p_OpsMagConvLD1AlmData1;
	p_tyLinkOpsMagConvLD2AlmData ACCESS p_OpsMagConvLD2AlmData;
	p_tyLinkOpsMagConvLD2AlmData1 ACCESS p_OpsMagConvLD2AlmData1;
	p_tyLinkOpsMagConvLD3AlmData ACCESS p_OpsMagConvLD3AlmData;
	p_tyLinkOpsMagConvLD3AlmData1 ACCESS p_OpsMagConvLD3AlmData1;
	p_tyLinkOpsMagConvLD4AlmData ACCESS p_OpsMagConvLD4AlmData;
	p_tyLinkOpsMagConvLD4AlmData1 ACCESS p_OpsMagConvLD4AlmData1;
	p_tyLinkSelClamp1AlmData ACCESS p_PneuNoSenSelClamp1AlmData;
	p_tyLinkSelClamp2AlmData ACCESS p_PneuNoSenSelClamp2AlmData;
	p_tyLinkSelClamp3AlmData ACCESS p_PneuNoSenSelClamp3AlmData;
	p_tyLinkSelClamp4AlmData ACCESS p_PneuNoSenSelClamp4AlmData;
	p_tyLinkUSSOT1AlmData ACCESS p_USSOT1AlmData;
	p_tyLinkUSSOT2AlmData ACCESS p_USSOT2AlmData;
	p_tyLinkUSSOT3AlmData ACCESS p_USSOT3AlmData;
	p_tyLinkUSSOT4AlmData ACCESS p_USSOT4AlmData;
	p_tyLinkDSSOT1AlmData ACCESS p_DSSOT1AlmData;
	p_tyLinkDSSOT2AlmData ACCESS p_DSSOT2AlmData;
	p_tyLinkDSSOT3AlmData ACCESS p_DSSOT3AlmData;
	p_tyLinkDSSOT4AlmData ACCESS p_DSSOT4AlmData;
	p_tyLinkMcAlarmData ACCESS p_McAlmData;
	p_tyLinkMc1AlarmData ACCESS p_Mc1AlmData;
	p_tyLinkUSBBarcodeAlmData ACCESS p_USBRdrAlmData;
	p_tyLinkUSBBarcodeAlmData1 ACCESS p_USBRdrAlmData1;
	p_tyLinkUSBBarcodeAlmData2 ACCESS p_USBRdrAlmData2;
	p_tyLinkAGVAlmData1 ACCESS p_AGVAlmData1;
	p_tyLinkRS232FrmAlmData ACCESS p_FrmAlmData;
	p_tyLinkAWPushOrPullerAlmData ACCESS p_AWPushOrPullerAlmData;
	p_tyLinkAWPushOrPullerAlmData1 ACCESS p_AWPushOrPullerAlmData1;
	p_tyLinkAWPushOrPullerAlmData2 ACCESS p_AWPushOrPullerAlmData2;
	p_tyLinkAWPushOrPullerAlmData3 ACCESS p_AWPushOrPullerAlmData3;
	p_tyLinkMtrPshrAlmData ACCESS p_MtrPshrAlmData;
//	p_tyLinkUSHermesInfoData1 ACCESS p_USHermesInfoData1;//new for Hermes 1.3
//	p_tyLinkUSHermesInfoData2 ACCESS p_USHermesInfoData2;//new for Hermes 1.3
	p_tyLinkRmtHermesInfoData ACCESS p_RmtHermesInfoData;//new for Hermes 1.3
	p_tyLinkSvyHermesAlmData ACCESS p_SvyHermesAlmData;//new for Hermes 1.3
	p_tyLinkSvyHermesAlmData1 ACCESS p_SvyHermesAlmData1;//new for Hermes 1.3
	p_tyLinkSvyHermesAlmData2 ACCESS p_SvyHermesAlmData2;//new for Hermes 1.3
	p_tyLinkSvyHermesAlmData3 ACCESS p_SvyHermesAlmData3;//new for Hermes 1.3
	p_tyLinkSvyHermesAlmData4 ACCESS p_SvyHermesAlmData4;//new for Hermes 1.3
	p_tyLinkSvyHermesInfoData ACCESS p_SvyHermesInfoData;//new for Hermes 1.3
	p_tyLinkSvyHermesInfoData1 ACCESS p_SvyHermesInfoData1;//new for Hermes 1.3
	p_tyLinkSvyHermesInfoData2 ACCESS p_SvyHermesInfoData2;//new for Hermes 1.3
	p_tyLinkSvyHermesInfoData3 ACCESS p_SvyHermesInfoData3;//new for Hermes 1.3
	p_tyLinkSvyHermesInfoData4 ACCESS p_SvyHermesInfoData4;//new for Hermes 1.3
	p_tyLinkOutShutterAlmData2 ACCESS p_Pneu2SenOutShutterAlmData2;
	p_tyLinkTrllyAlmData ACCESS p_PneuExtSenTrllyAlmData;
	p_tyLinkTrlly2AlmData ACCESS p_PneuExtSenTrlly2AlmData;

	p_tyLinkOpsLifMagLDAlmData ACCESS p_OpsLifMagLDAlmData;
	p_tyLinkOpsLifMagLDAlmData1 ACCESS p_OpsLifMagLDAlmData1;

	p_tyLinkPPAlmData ACCESS p_PPAlmData;
	p_tyLinkPPAlmData1 ACCESS p_PPAlmData1;
	p_tyLinkPPAlmData2 ACCESS p_PPAlmData2;
	p_tyLinkPPAlmData3 ACCESS p_PPAlmData3;

	p_tyLinkInShutterAlmData2 ACCESS p_Pneu2SenInShutterAlmData2;
	p_tyLinkInShutterAlmData3 ACCESS p_Pneu2SenInShutterAlmData3;

	p_tyLinkAutoRcpAlmData ACCESS p_AutoRcpAlmData;
	p_tyLinkAutoRcpInfoData ACCESS p_AutoRcpInfoData;
	p_tyLinkAutoRcpInfoData1 ACCESS p_AutoRcpInfoData1;

	//Pass Data To Internal Use
	p_udiRstErr ACCESS p_RstErrReset;
	p_eAct ACCESS p_StartupAlarmAct;
	p_dtCurrDT ACCESS p_TimeCurrDT;
	p_udiFileKeepDay ACCESS p_NtParamAlmFileKeepDay;
	p_sProgNm ACCESS p_NtParamAlmProgNm;
	p_bNtSettingsLoadDone ACCESS p_StartupNtSettingsLoadDone;
	p_bStartupUISettingsLoadDone ACCESS p_StartupUISettingsLoadDone;
	(* Always Change If Project Change *)

END_ACTION
```

#### Act_Initial.st
```iecst
(** 2019-01-03 **)
ACTION Act_Initial:

	//Initial
	sStatTxt	:= a_sStatText[eStat];

	fbDirCreate1.sDevice	:= 'F';
	fbDirCreate1.sDirName	:= 'User';
	fbDirCreate1(bEn := FALSE);

	fbDirCreate2.sDevice	:= 'User';
	fbDirCreate2.sDirName	:= 'Alarm';
	fbDirCreate2(bEn := FALSE);

	fbFileAppend1.sDevice	:= 'Alarm';
	fbFileAppend1(bEn := FALSE);

	fbFileOldDel1.sDevice	:= 'Alarm';
	fbFileOldDel1.sPath		:= '';
	fbFileOldDel1.sKeyword	:= 'ALARM_';
	fbFileOldDel1(bEn := FALSE);

	fbFileRead1.sDevice		:= 'Alarm';
	fbFileRead1.sFile		:= 'History.dat';
	fbFileRead1.udiOffset	:= 0;
	fbFileRead1.p_Dest		:= ADR(a_sHistoryList);
	fbFileRead1.udiLen		:= SIZEOF(a_sHistoryList);
	fbFileRead1(bEn := FALSE);

	fbFileWrite1.sDevice	:= 'Alarm';
	fbFileWrite1.sFile		:= 'History.dat';
	fbFileWrite1.udiOffset	:= 0;
	fbFileWrite1.p_Src		:= ADR(a_sHistoryList);
	fbFileWrite1.udiLen		:= SIZEOF(a_sHistoryList);
	fbFileWrite1.udiOption	:= 0;
	fbFileWrite1(bEn := FALSE);

END_ACTION
```
